   VAR
      sFB_ParaAcycRead { ExternalAccessible := 'False'; ExternalVisible := 'False'; ExternalWritable := 'False'; S7_SetPoint := 'False'} : "FB_VfdNORDParaAcycRead";
      sFB_ParaAcycWrite { ExternalAccessible := 'False'; ExternalVisible := 'False'; ExternalWritable := 'False'; S7_SetPoint := 'False'} : "FB_VfdNORDParaAcycWrite";
      sR_TRIG_Done {InstructionName := 'R_TRIG'; LibVersion := '1.0'; ExternalAccessible := 'False'; ExternalVisible := 'False'; ExternalWritable := 'False'; S7_SetPoint := 'False'} : R_TRIG;
      sR_TRIG_StartJob {InstructionName := 'R_TRIG'; LibVersion := '1.0'; ExternalAccessible := 'False'; ExternalVisible := 'False'; ExternalWritable := 'False'; S7_SetPoint := 'False'} : R_TRIG;   // Bit for start trigger for rising edge
      sF_TRIG_CancelJob {InstructionName := 'F_TRIG'; LibVersion := '1.0'; ExternalAccessible := 'False'; ExternalVisible := 'False'; ExternalWritable := 'False'; S7_SetPoint := 'False'} : F_TRIG;   // Bit for start trigger for falling edge
      sa_Parameter { ExternalAccessible := 'False'; ExternalVisible := 'False'; ExternalWritable := 'False'; S7_SetPoint := 'False'} : Array[0..60] of "UDT_VfdNordParameter";   // Data of parameters
      sa_Status { ExternalAccessible := 'False'; ExternalVisible := 'False'; ExternalWritable := 'False'} : Struct   // Parametrization status
         StepNrError { ExternalAccessible := 'False'; ExternalVisible := 'False'; ExternalWritable := 'False'} : Int;   // The number of the step in witch the error occurred
         ParameterNrError { ExternalAccessible := 'False'; ExternalVisible := 'False'; ExternalWritable := 'False'} : Int;   // The number of the parameter in witch the error occurred
         StepNr { ExternalAccessible := 'False'; ExternalVisible := 'False'; ExternalWritable := 'False'} : Int := 0;   // Current step number
         ResponseValueError { ExternalAccessible := 'False'; ExternalVisible := 'False'; ExternalWritable := 'False'} : Bool;   // Response value error
         WrongFormat { ExternalAccessible := 'False'; ExternalVisible := 'False'; ExternalWritable := 'False'} : Bool;   // Wrong parameter format
         TimeExceeded { ExternalAccessible := 'False'; ExternalVisible := 'False'; ExternalWritable := 'False'} : Bool;   // Time has been exceeded
         NeedAck { ExternalAccessible := 'False'; ExternalVisible := 'False'; ExternalWritable := 'False'} : Bool;   // Need acknowledge signal (to cintinue parametrization)
         StepDone { ExternalAccessible := 'False'; ExternalVisible := 'False'; ExternalWritable := 'False'} : Bool;   // Step done
      END_STRUCT;
      si_StepTime { ExternalAccessible := 'False'; ExternalVisible := 'False'; ExternalWritable := 'False'} : Int;
      si_StepMax { ExternalAccessible := 'False'; ExternalVisible := 'False'; ExternalWritable := 'False'} : Int := 0;   // Maximum step number
      sx_Start { ExternalAccessible := 'False'; ExternalVisible := 'False'; ExternalWritable := 'False'} : Bool;   // Signal to start of parameterization function SinaPara
      sx_Busy { ExternalAccessible := 'False'; ExternalVisible := 'False'; ExternalWritable := 'False'} : Bool;   // Parametrization in progress (busy)
      sx_Done { ExternalAccessible := 'False'; ExternalVisible := 'False'; ExternalWritable := 'False'} : Bool;   // Parametrization done
      sx_Error { ExternalAccessible := 'False'; ExternalVisible := 'False'; ExternalWritable := 'False'} : Bool;   // Main error signal
      sx_PreparedData { ExternalAccessible := 'False'; ExternalVisible := 'False'; ExternalWritable := 'False'} : Bool;   // Step data prepared
      sx_ReadOrder { ExternalAccessible := 'False'; ExternalVisible := 'False'; ExternalWritable := 'False'} : Bool;   // Order to read paraeter with transition from 0 to 1
      sx_WriteOrder { ExternalAccessible := 'False'; ExternalVisible := 'False'; ExternalWritable := 'False'} : Bool;   // Order to write parameter with transition from 0 to 1
      sx_MaxStepCalculation { ExternalAccessible := 'False'; ExternalVisible := 'False'; ExternalWritable := 'False'} : Bool;   // Maximum step calculated
   END_VAR
   VAR RETAIN
      sx_24VCommissioningDone { ExternalAccessible := 'False'; ExternalVisible := 'False'; ExternalWritable := 'False'} : Bool;   // 24V commissioning done succesfully
   END_VAR

   VAR_TEMP
      ti_index : Int;   // Temporary array index
      ti_ControlMethod : Int;
      ti_EncoderCode : Int;
      ti_i : Int;   // Loop counter
      ti_BrakeReaction : Int;
   END_VAR

   VAR CONSTANT
      ci_CFC_ClosedLoop : Int := 1;
      ci_CFC_OpenLoop : Int := 0;
      ci_EncoderRes512 : Int := 1;
      ci_EncoderRes1024 : Int := 3;
      ci_EncoderRes2048 : Int := 5;
      ci_EncoderRes4096 : Int := 6;
      ci_MaxStepTime : Int := 100;
   END_VAR


BEGIN
	(*
	----------------------------------------------------------------------------------------

	Version history:
	Date        | Version   | Author        | Remark
	----------------------------------------------------------------------------------------
	12/01/2020  | 0.1       | S.Theocharis  | Initial version TIA 15.1
	08/04/2021  | 0.2       | F.Baten       | New read/write blocks
	                                        | New motor parameter set ( most values not 32bit )
	                                        | PN device with onboard safety
	                                        | Reading and writing optimised
	27/01/2022  | 0.3       | K.Pokorski    | Add 24V and 400V commissionig status
	                                        | Fix VFD Output bug
	                                        | Initialize InUse status in all parameters
	                                        | Fix Motor identification
	                                        | Save parameters to External memory
	                                        | Delete saving F-parameters from sequence (not working and creating faults)
	                                        | Delete reading CRC code (reading old CRC code what can be confusing)
	21/04/2022  | 0.4       | K.Pokorski    | Delete motor identification
	21/02/2023  | 4.0       | F.Baten       | 4.0 Release TIA 17.5

	*)

	REGION 1 - Start Job

	    // Monitor rising trigger if is input enable signal
	    #sR_TRIG_StartJob(CLK := #iqx_Enable);

	    IF (#sR_TRIG_StartJob.Q)
	    THEN
	        #sx_Start := TRUE;
	        #sx_Busy := TRUE;
	        #sx_Done := FALSE;
	        #sx_Error := FALSE;
	        #sx_PreparedData := FALSE;
	        #sx_MaxStepCalculation := FALSE;
	        #sa_Status.StepDone := FALSE;
	        #sa_Status.StepNrError := 0;
	        #sa_Status.ParameterNrError := 0;
	        #sa_Status.StepNr := 0;
	        #si_StepTime := 0;
	        #qi_HWAdress := 0;

	        FOR #ti_i := 0 TO 60 DO
	            #sa_Parameter[#ti_i].InUse := FALSE;
	        END_FOR;



	    END_IF;

	END_REGION

	REGION 2 - Build Sequences in static memory

	    IF #sR_TRIG_StartJob.Q THEN
	        //  IF NOT #sx_24VCommissioningDone THEN
	        REGION Step 01 - P523 Factory reset [0..3]
	            #ti_index := 0;
	            #sa_Parameter[#ti_index].ParaNumber := 523;
	            #sa_Parameter[#ti_index].Index := 0;
	            #sa_Parameter[#ti_index].WriteValue := 1;
	            #sa_Parameter[#ti_index].WriteAccess := TRUE;
	            #sa_Parameter[#ti_index].ParaSet := 0;
	            #sa_Parameter[#ti_index].Format32 := FALSE;
	            #sa_Parameter[#ti_index].ActualValue := 0;
	            #sa_Parameter[#ti_index].InUse := TRUE;
	            #sa_Parameter[#ti_index].RamOnly := FALSE;
	        END_REGION

	        REGION Step 02 - P003 Set supervisor code to access all parameters [0..9999]
	            #ti_index := #ti_index + 1;
	            #sa_Parameter[#ti_index].ParaNumber := 3;
	            #sa_Parameter[#ti_index].Index := 0;
	            #sa_Parameter[#ti_index].WriteValue := 3;
	            #sa_Parameter[#ti_index].WriteAccess := TRUE;
	            #sa_Parameter[#ti_index].ParaSet := 0;
	            #sa_Parameter[#ti_index].Format32 := FALSE;
	            #sa_Parameter[#ti_index].ActualValue := 0;
	            #sa_Parameter[#ti_index].InUse := TRUE;
	            #sa_Parameter[#ti_index].RamOnly := FALSE;
	        END_REGION

	        REGION Step 03 - P800 Set Operating mode Safety [0-1]
	            #ti_index := #ti_index + 1;
	            #sa_Parameter[#ti_index].ParaNumber := 800;
	            #sa_Parameter[#ti_index].Index := 1;
	            #sa_Parameter[#ti_index].WriteValue := 1;
	            #sa_Parameter[#ti_index].WriteAccess := TRUE;
	            #sa_Parameter[#ti_index].ParaSet := 0;
	            #sa_Parameter[#ti_index].Format32 := FALSE;
	            #sa_Parameter[#ti_index].ActualValue := 0;
	            #sa_Parameter[#ti_index].InUse := TRUE;
	            #sa_Parameter[#ti_index].RamOnly := FALSE;
	        END_REGION

	        REGION Step 04 - P800 Set Operating mode Safety [0-1]
	            #ti_index := #ti_index + 1;
	            #sa_Parameter[#ti_index].ParaNumber := 800;
	            #sa_Parameter[#ti_index].Index := 2;
	            #sa_Parameter[#ti_index].WriteValue := 0;
	            #sa_Parameter[#ti_index].WriteAccess := TRUE;
	            #sa_Parameter[#ti_index].ParaSet := 0;
	            #sa_Parameter[#ti_index].Format32 := FALSE;
	            #sa_Parameter[#ti_index].ActualValue := 0;
	            #sa_Parameter[#ti_index].InUse := TRUE;
	            #sa_Parameter[#ti_index].RamOnly := FALSE;
	        END_REGION

	        REGION Step 05 - P802 Set Enable safety channel [0-1]  Channel 1 on
	            #ti_index := #ti_index + 1;
	            #sa_Parameter[#ti_index].ParaNumber := 802;
	            #sa_Parameter[#ti_index].Index := 1;
	            #sa_Parameter[#ti_index].WriteValue := 1;
	            #sa_Parameter[#ti_index].WriteAccess := TRUE;
	            #sa_Parameter[#ti_index].ParaSet := 0;
	            #sa_Parameter[#ti_index].Format32 := FALSE;
	            #sa_Parameter[#ti_index].ActualValue := 0;
	            #sa_Parameter[#ti_index].InUse := TRUE;
	            #sa_Parameter[#ti_index].RamOnly := FALSE;
	        END_REGION

	        REGION Step 06 - P802 Set Enable safety channel [0-1]  Channel 2 on
	            #ti_index := #ti_index + 1;
	            #sa_Parameter[#ti_index].ParaNumber := 802;
	            #sa_Parameter[#ti_index].Index := 2;
	            #sa_Parameter[#ti_index].WriteValue := 1;
	            #sa_Parameter[#ti_index].WriteAccess := TRUE;
	            #sa_Parameter[#ti_index].ParaSet := 0;
	            #sa_Parameter[#ti_index].Format32 := FALSE;
	            #sa_Parameter[#ti_index].ActualValue := 0;
	            #sa_Parameter[#ti_index].InUse := TRUE;
	            #sa_Parameter[#ti_index].RamOnly := FALSE;
	        END_REGION

	        REGION Step 07 - P802 Set Enable safety channel [0-1]  Channel 3 on
	            #ti_index := #ti_index + 1;
	            #sa_Parameter[#ti_index].ParaNumber := 802;
	            #sa_Parameter[#ti_index].Index := 3;
	            #sa_Parameter[#ti_index].WriteValue := 1;
	            #sa_Parameter[#ti_index].WriteAccess := TRUE;
	            #sa_Parameter[#ti_index].ParaSet := 0;
	            #sa_Parameter[#ti_index].Format32 := FALSE;
	            #sa_Parameter[#ti_index].ActualValue := 0;
	            #sa_Parameter[#ti_index].InUse := TRUE;
	            #sa_Parameter[#ti_index].RamOnly := FALSE;
	        END_REGION

	        REGION Step 08 - P846 Read dipswitches
	            #ti_index := #ti_index + 1;
	            #sa_Parameter[#ti_index].ParaNumber := 846;
	            #sa_Parameter[#ti_index].Index := 0;
	            #sa_Parameter[#ti_index].WriteValue := 0;
	            #sa_Parameter[#ti_index].WriteAccess := FALSE;
	            #sa_Parameter[#ti_index].ParaSet := 0;
	            #sa_Parameter[#ti_index].Format32 := FALSE;
	            #sa_Parameter[#ti_index].ActualValue := 0;
	            #sa_Parameter[#ti_index].InUse := TRUE;
	            #sa_Parameter[#ti_index].RamOnly := FALSE;
	        END_REGION

	        REGION Step 09 - P120 Set extern control units [0-1]  Switch off 3 and 4
	            #ti_index := #ti_index + 1;
	            #sa_Parameter[#ti_index].ParaNumber := 120;
	            #sa_Parameter[#ti_index].Index := 3;
	            #sa_Parameter[#ti_index].WriteValue := 0;
	            #sa_Parameter[#ti_index].WriteAccess := TRUE;
	            #sa_Parameter[#ti_index].ParaSet := 0;
	            #sa_Parameter[#ti_index].Format32 := FALSE;
	            #sa_Parameter[#ti_index].ActualValue := 0;
	            #sa_Parameter[#ti_index].InUse := TRUE;
	            #sa_Parameter[#ti_index].RamOnly := FALSE;
	        END_REGION

	        REGION Step 10 - P120 Set extern control units [0-1]  Switch off 3 and 4
	            #ti_index := #ti_index + 1;
	            #sa_Parameter[#ti_index].ParaNumber := 120;
	            #sa_Parameter[#ti_index].Index := 4;
	            #sa_Parameter[#ti_index].WriteValue := 0;
	            #sa_Parameter[#ti_index].WriteAccess := TRUE;
	            #sa_Parameter[#ti_index].ParaSet := 0;
	            #sa_Parameter[#ti_index].Format32 := FALSE;
	            #sa_Parameter[#ti_index].ActualValue := 0;
	            #sa_Parameter[#ti_index].InUse := TRUE;
	            #sa_Parameter[#ti_index].RamOnly := FALSE;
	        END_REGION

	        REGION Step 11 - P202 Write motor nominal speed [150...24000]rpm
	            #ti_index := #ti_index + 1;
	            #sa_Parameter[#ti_index].ParaNumber := 202;
	            #sa_Parameter[#ti_index].Index := 0;
	            #sa_Parameter[#ti_index].WriteValue := #iudt_MotorData.NominalSpeed;
	            #sa_Parameter[#ti_index].WriteAccess := TRUE;
	            #sa_Parameter[#ti_index].ParaSet := 1; // Parameter set 1
	            #sa_Parameter[#ti_index].Format32 := FALSE;
	            #sa_Parameter[#ti_index].ActualValue := 0;
	            #sa_Parameter[#ti_index].InUse := TRUE;
	            #sa_Parameter[#ti_index].RamOnly := FALSE;
	        END_REGION

	        REGION Step 12 - P203 Write motor nominal current [0.1 ...1000.0]A
	            #ti_index := #ti_index + 1;
	            #sa_Parameter[#ti_index].ParaNumber := 203;
	            #sa_Parameter[#ti_index].Index := 0;
	            #sa_Parameter[#ti_index].WriteValue := (REAL_TO_DINT(#iudt_MotorData.NominalCurrent * 10));  // Value 55 = 5.5 Amps
	            #sa_Parameter[#ti_index].WriteAccess := TRUE;
	            #sa_Parameter[#ti_index].ParaSet := 0; // Parameter set 1
	            #sa_Parameter[#ti_index].Format32 := FALSE;
	            #sa_Parameter[#ti_index].ActualValue := 0;
	            #sa_Parameter[#ti_index].InUse := TRUE;
	            #sa_Parameter[#ti_index].RamOnly := FALSE;
	        END_REGION

	        REGION Step 13 - P204 Write motor nominal voltage [100 ... 800]V
	            #ti_index := #ti_index + 1;
	            #sa_Parameter[#ti_index].ParaNumber := 204;
	            #sa_Parameter[#ti_index].Index := 0;
	            #sa_Parameter[#ti_index].WriteValue := #iudt_MotorData.NominalVoltage;
	            #sa_Parameter[#ti_index].WriteAccess := FALSE;
	            #sa_Parameter[#ti_index].ParaSet := 1; // Parameter set 1
	            #sa_Parameter[#ti_index].Format32 := FALSE;
	            #sa_Parameter[#ti_index].ActualValue := 0;
	            #sa_Parameter[#ti_index].InUse := TRUE;
	            #sa_Parameter[#ti_index].RamOnly := FALSE;
	        END_REGION

	        REGION Step 14 - P205 Write motor nominal power
	            #ti_index := #ti_index + 1;
	            #sa_Parameter[#ti_index].ParaNumber := 205;
	            #sa_Parameter[#ti_index].Index := 0;
	            #sa_Parameter[#ti_index].WriteValue := (REAL_TO_DINT(#iudt_MotorData.NominalPower * 100));
	            #sa_Parameter[#ti_index].WriteAccess := TRUE;
	            #sa_Parameter[#ti_index].ParaSet := 0; // Parameter set 1
	            #sa_Parameter[#ti_index].Format32 := FALSE;
	            #sa_Parameter[#ti_index].ActualValue := 0;
	            #sa_Parameter[#ti_index].InUse := TRUE;
	            #sa_Parameter[#ti_index].RamOnly := FALSE;
	        END_REGION

	        REGION Step 15 - P206 Write motor cosPhi [0.50 ... 0.95]
	            #ti_index := #ti_index + 1;
	            #sa_Parameter[#ti_index].ParaNumber := 206;
	            #sa_Parameter[#ti_index].Index := 0;
	            #sa_Parameter[#ti_index].WriteValue := REAL_TO_DINT(#iudt_MotorData.CosPhi * 100);
	            #sa_Parameter[#ti_index].WriteAccess := TRUE;
	            #sa_Parameter[#ti_index].ParaSet := 0; // Parameter set 1
	            #sa_Parameter[#ti_index].Format32 := FALSE;
	            #sa_Parameter[#ti_index].ActualValue := 0;
	            #sa_Parameter[#ti_index].InUse := TRUE;
	            #sa_Parameter[#ti_index].RamOnly := FALSE;
	        END_REGION

	        REGION Step 16 - P207 Connection Star / Delta [0=Star 1=Delta]
	            #ti_index := #ti_index + 1;
	            #sa_Parameter[#ti_index].ParaNumber := 207;
	            #sa_Parameter[#ti_index].Index := 0;
	            #sa_Parameter[#ti_index].WriteValue := #iudt_MotorData.Connection;
	            #sa_Parameter[#ti_index].WriteAccess := TRUE;
	            #sa_Parameter[#ti_index].ParaSet := 0; // Parameter set 1
	            #sa_Parameter[#ti_index].Format32 := FALSE;
	            #sa_Parameter[#ti_index].ActualValue := 0;
	            #sa_Parameter[#ti_index].InUse := TRUE;
	            #sa_Parameter[#ti_index].RamOnly := FALSE;
	        END_REGION

	        REGION Step 17 - P105 Write Maximum / Reference Frequency [0.1...400.0]Hz
	            #ti_index := #ti_index + 1;
	            #sa_Parameter[#ti_index].ParaNumber := 105;
	            #sa_Parameter[#ti_index].Index := 0;
	            #sa_Parameter[#ti_index].WriteValue := REAL_TO_DINT(#ir_ReferenceFrequency * 10);
	            #sa_Parameter[#ti_index].WriteAccess := TRUE;
	            #sa_Parameter[#ti_index].ParaSet := 0; // Parameter set 1
	            #sa_Parameter[#ti_index].Format32 := FALSE;
	            #sa_Parameter[#ti_index].ActualValue := 0;
	            #sa_Parameter[#ti_index].InUse := TRUE;
	            #sa_Parameter[#ti_index].RamOnly := FALSE;
	        END_REGION

	        REGION Step 18 - P107 Brake reaction
	            IF #iudt_MotorData.BrakeConfig THEN
	                #ti_BrakeReaction := 20;
	            ELSE
	                #ti_BrakeReaction := 0;
	            END_IF;

	            #ti_index := #ti_index + 1;
	            #sa_Parameter[#ti_index].ParaNumber := 107;
	            #sa_Parameter[#ti_index].Index := 0;
	            #sa_Parameter[#ti_index].WriteValue := #ti_BrakeReaction;
	            #sa_Parameter[#ti_index].WriteAccess := TRUE;
	            #sa_Parameter[#ti_index].ParaSet := 0; // Parameter set 1
	            #sa_Parameter[#ti_index].Format32 := FALSE;
	            #sa_Parameter[#ti_index].ActualValue := 0;
	            #sa_Parameter[#ti_index].InUse := TRUE;
	            #sa_Parameter[#ti_index].RamOnly := FALSE;
	        END_REGION

	        REGION Step 19 - P300 Mode [0..2]
	            //If an IE4 motor is operated in CFC closed loop mode , the slip error monitoring must be activated. P327<>0
	            IF #iudt_MotorData.EncoderResolution <> 0 THEN
	                #ti_ControlMethod := #ci_CFC_ClosedLoop; //CFC closed loop control. Speed control with encoder feedback
	            ELSE
	                #ti_ControlMethod := #ci_CFC_OpenLoop; //VFC open loop control. Speed control without encoder feedback
	            END_IF;
	            #ti_index := #ti_index + 1;
	            #sa_Parameter[#ti_index].ParaNumber := 300;
	            #sa_Parameter[#ti_index].Index := 0;
	            #sa_Parameter[#ti_index].WriteValue := #ti_ControlMethod;
	            #sa_Parameter[#ti_index].WriteAccess := TRUE;
	            #sa_Parameter[#ti_index].ParaSet := 1; // Parameter set 1
	            #sa_Parameter[#ti_index].Format32 := FALSE;
	            #sa_Parameter[#ti_index].ActualValue := 0;
	            #sa_Parameter[#ti_index].InUse := TRUE;
	            #sa_Parameter[#ti_index].RamOnly := FALSE;
	        END_REGION

	        REGION Step 20 - P301 Encoder Resolution [0..17]
	            CASE #iudt_MotorData.EncoderResolution OF
	                512:
	                    #ti_EncoderCode := #ci_EncoderRes512;
	                1024:
	                    #ti_EncoderCode := #ci_EncoderRes1024;
	                2048:
	                    #ti_EncoderCode := #ci_EncoderRes2048;
	                4096:
	                    #ti_EncoderCode := #ci_EncoderRes4096;
	                ELSE
	                    #ti_EncoderCode := 6; //default value
	            END_CASE;

	            #ti_index := #ti_index + 1;
	            #sa_Parameter[#ti_index].ParaNumber := 301;
	            #sa_Parameter[#ti_index].Index := 0;
	            #sa_Parameter[#ti_index].WriteValue := #ti_EncoderCode;
	            #sa_Parameter[#ti_index].WriteAccess := TRUE;
	            #sa_Parameter[#ti_index].ParaSet := 0;
	            #sa_Parameter[#ti_index].Format32 := FALSE;
	            #sa_Parameter[#ti_index].ActualValue := 0;
	            #sa_Parameter[#ti_index].InUse := TRUE;
	            #sa_Parameter[#ti_index].RamOnly := FALSE;
	        END_REGION

	        REGION Step 21 - P326 Encoder ratio [0.01 ... 100.0]
	            #ti_index := #ti_index + 1;
	            #sa_Parameter[#ti_index].ParaNumber := 326;
	            #sa_Parameter[#ti_index].Index := 0;
	            #sa_Parameter[#ti_index].WriteValue := (1 * 100); //leave temporary the default 1.00;
	            #sa_Parameter[#ti_index].WriteAccess := TRUE;
	            #sa_Parameter[#ti_index].ParaSet := 0;
	            #sa_Parameter[#ti_index].Format32 := FALSE;
	            #sa_Parameter[#ti_index].ActualValue := 0;
	            #sa_Parameter[#ti_index].InUse := TRUE;
	            #sa_Parameter[#ti_index].RamOnly := FALSE;
	        END_REGION

	        REGION Step 22 - P420[1] Digital inputs [0 ... 80] DI1
	            #ti_index := #ti_index + 1;
	            #sa_Parameter[#ti_index].ParaNumber := 420;
	            #sa_Parameter[#ti_index].Index := 1;
	            #sa_Parameter[#ti_index].WriteValue := 0;
	            #sa_Parameter[#ti_index].WriteAccess := TRUE;
	            #sa_Parameter[#ti_index].ParaSet := 0;
	            #sa_Parameter[#ti_index].Format32 := FALSE;
	            #sa_Parameter[#ti_index].ActualValue := 0;
	            #sa_Parameter[#ti_index].InUse := TRUE;
	            #sa_Parameter[#ti_index].RamOnly := FALSE;
	        END_REGION

	        REGION Step 23 - P420[2] Digital inputs [0 ... 80] DI2
	            #ti_index := #ti_index + 1;
	            #sa_Parameter[#ti_index].ParaNumber := 420;
	            #sa_Parameter[#ti_index].Index := 2;
	            #sa_Parameter[#ti_index].WriteValue := 0;
	            #sa_Parameter[#ti_index].WriteAccess := TRUE;
	            #sa_Parameter[#ti_index].ParaSet := 0;
	            #sa_Parameter[#ti_index].Format32 := FALSE;
	            #sa_Parameter[#ti_index].ActualValue := 0;
	            #sa_Parameter[#ti_index].InUse := TRUE;
	            #sa_Parameter[#ti_index].RamOnly := FALSE;
	        END_REGION

	        REGION Step 24 - P420[3] Digital inputs [0 ... 80] DI3
	            #ti_index := #ti_index + 1;
	            #sa_Parameter[#ti_index].ParaNumber := 420;
	            #sa_Parameter[#ti_index].Index := 3;
	            #sa_Parameter[#ti_index].WriteValue := 0;
	            #sa_Parameter[#ti_index].WriteAccess := TRUE;
	            #sa_Parameter[#ti_index].ParaSet := 0;
	            #sa_Parameter[#ti_index].Format32 := FALSE;
	            #sa_Parameter[#ti_index].ActualValue := 0;
	            #sa_Parameter[#ti_index].InUse := TRUE;
	            #sa_Parameter[#ti_index].RamOnly := FALSE;
	        END_REGION

	        REGION Step 25 - P426 Quick Stop time [0 ... 320.00] sec
	            #ti_index := #ti_index + 1;
	            #sa_Parameter[#ti_index].ParaNumber := 426;
	            #sa_Parameter[#ti_index].Index := 0;
	            #sa_Parameter[#ti_index].WriteValue := 60;
	            #sa_Parameter[#ti_index].WriteAccess := TRUE;
	            #sa_Parameter[#ti_index].ParaSet := 1; //paraset 1
	            #sa_Parameter[#ti_index].Format32 := FALSE;
	            #sa_Parameter[#ti_index].ActualValue := 0;
	            #sa_Parameter[#ti_index].InUse := TRUE;
	            #sa_Parameter[#ti_index].RamOnly := FALSE;
	        END_REGION

	        REGION Step 26 - P509 Control word source [0..4]
	            #ti_index := #ti_index + 1;
	            #sa_Parameter[#ti_index].ParaNumber := 509;
	            #sa_Parameter[#ti_index].Index := 0;
	            #sa_Parameter[#ti_index].WriteValue := 3; // System bus communication (PN)
	            #sa_Parameter[#ti_index].WriteAccess := TRUE;
	            #sa_Parameter[#ti_index].ParaSet := 0;
	            #sa_Parameter[#ti_index].Format32 := FALSE;
	            #sa_Parameter[#ti_index].ActualValue := 0;
	            #sa_Parameter[#ti_index].InUse := TRUE;
	            #sa_Parameter[#ti_index].RamOnly := FALSE;
	        END_REGION

	        REGION Step 27 - P543[1] Actual speed to actual value 1 [0..57]
	            #ti_index := #ti_index + 1;
	            #sa_Parameter[#ti_index].ParaNumber := 543;
	            #sa_Parameter[#ti_index].Index := 1;
	            #sa_Parameter[#ti_index].WriteValue := 1; // 2 = Set Actual value 1 to actual speed
	            #sa_Parameter[#ti_index].WriteAccess := TRUE;
	            #sa_Parameter[#ti_index].ParaSet := 1; // Parameter set 1
	            #sa_Parameter[#ti_index].Format32 := FALSE;
	            #sa_Parameter[#ti_index].ActualValue := 0;
	            #sa_Parameter[#ti_index].InUse := TRUE;
	            #sa_Parameter[#ti_index].RamOnly := FALSE;
	        END_REGION

	        REGION Step 28 - P543[2] Error code to actual value 2 [0..57]
	            #ti_index := #ti_index + 1;
	            #sa_Parameter[#ti_index].ParaNumber := 543;
	            #sa_Parameter[#ti_index].Index := 2;
	            #sa_Parameter[#ti_index].WriteValue := 9; // 9 =  Set Actual value 2 to error code
	            #sa_Parameter[#ti_index].WriteAccess := TRUE;
	            #sa_Parameter[#ti_index].ParaSet := 1; // Parameter set 1
	            #sa_Parameter[#ti_index].Format32 := FALSE;
	            #sa_Parameter[#ti_index].ActualValue := 0;
	            #sa_Parameter[#ti_index].InUse := TRUE;
	            #sa_Parameter[#ti_index].RamOnly := FALSE;
	        END_REGION

	        REGION Step 29 - P543[3] DIO status to actual value 3 [0..57]
	            #ti_index := #ti_index + 1;
	            #sa_Parameter[#ti_index].ParaNumber := 543;
	            #sa_Parameter[#ti_index].Index := 3;
	            #sa_Parameter[#ti_index].WriteValue := 5; // 5 =  Set Actual value 3 to DIO status
	            #sa_Parameter[#ti_index].WriteAccess := TRUE;
	            #sa_Parameter[#ti_index].ParaSet := 1; // Parameter set 1
	            #sa_Parameter[#ti_index].Format32 := FALSE;
	            #sa_Parameter[#ti_index].ActualValue := 0;
	            #sa_Parameter[#ti_index].InUse := TRUE;
	            #sa_Parameter[#ti_index].RamOnly := FALSE;
	        END_REGION

	        REGION Step 30 - P546[1] Frequency setpoint to setpoint 1 [0..36]
	            #ti_index := #ti_index + 1;
	            #sa_Parameter[#ti_index].ParaNumber := 546;
	            #sa_Parameter[#ti_index].Index := 1;
	            #sa_Parameter[#ti_index].WriteValue := 1; // 5 =  Set setpoint 1 to frequency setpoint
	            #sa_Parameter[#ti_index].WriteAccess := TRUE;
	            #sa_Parameter[#ti_index].ParaSet := 1; // Parameter set 1
	            #sa_Parameter[#ti_index].Format32 := FALSE;
	            #sa_Parameter[#ti_index].ActualValue := 0;
	            #sa_Parameter[#ti_index].InUse := TRUE;
	            #sa_Parameter[#ti_index].RamOnly := FALSE;
	        END_REGION

	        REGION Step 31 - P546[2] Ramp setpoint to setpoint 2 [0..36]
	            #ti_index := #ti_index + 1;
	            #sa_Parameter[#ti_index].ParaNumber := 546;
	            #sa_Parameter[#ti_index].Index := 2;
	            #sa_Parameter[#ti_index].WriteValue := 15; // 15 =  Set setpoint 2 to ramp setpoint
	            #sa_Parameter[#ti_index].WriteAccess := TRUE;
	            #sa_Parameter[#ti_index].ParaSet := 1; // Parameter set 1
	            #sa_Parameter[#ti_index].Format32 := FALSE;
	            #sa_Parameter[#ti_index].ActualValue := 0;
	            #sa_Parameter[#ti_index].InUse := TRUE;
	            #sa_Parameter[#ti_index].RamOnly := FALSE;
	        END_REGION

	        REGION Step 32 - P546[3] DO control to setpoint 3 [0..36]
	            #ti_index := #ti_index + 1;
	            #sa_Parameter[#ti_index].ParaNumber := 546;
	            #sa_Parameter[#ti_index].Index := 3;
	            #sa_Parameter[#ti_index].WriteValue := 31; // 5 =  Set setpoint 3 to DIO
	            #sa_Parameter[#ti_index].WriteAccess := TRUE;
	            #sa_Parameter[#ti_index].ParaSet := 1; // Parameter set 1
	            #sa_Parameter[#ti_index].Format32 := FALSE;
	            #sa_Parameter[#ti_index].ActualValue := 0;
	            #sa_Parameter[#ti_index].InUse := TRUE;
	            #sa_Parameter[#ti_index].RamOnly := FALSE;
	        END_REGION

	        REGION Step 33 - P434[3] DO Function [1..2]
	            #ti_index := #ti_index + 1;
	            #sa_Parameter[#ti_index].ParaNumber := 434;
	            #sa_Parameter[#ti_index].Index := 1;
	            #sa_Parameter[#ti_index].WriteValue := 38;
	            #sa_Parameter[#ti_index].WriteAccess := TRUE;
	            #sa_Parameter[#ti_index].ParaSet := 1; // Parameter set 1
	            #sa_Parameter[#ti_index].Format32 := FALSE;
	            #sa_Parameter[#ti_index].ActualValue := 0;
	            #sa_Parameter[#ti_index].InUse := TRUE;
	            #sa_Parameter[#ti_index].RamOnly := FALSE;
	        END_REGION

	        REGION Step 34 - P560 Save [0..2]
	            #ti_index := #ti_index + 1;
	            #sa_Parameter[#ti_index].ParaNumber := 560;
	            #sa_Parameter[#ti_index].Index := 0;
	            #sa_Parameter[#ti_index].WriteValue := 1; // 1= save RAM & EERPOM
	            #sa_Parameter[#ti_index].WriteAccess := TRUE;
	            #sa_Parameter[#ti_index].ParaSet := 0;
	            #sa_Parameter[#ti_index].Format32 := FALSE;
	            #sa_Parameter[#ti_index].ActualValue := 0;
	            #sa_Parameter[#ti_index].InUse := TRUE;
	            #sa_Parameter[#ti_index].RamOnly := FALSE;
	        END_REGION

	        REGION Step 35 - P550 Copy internal EEPROM to external EEPROM [0..3]
	            #ti_index := #ti_index + 1;
	            #sa_Parameter[#ti_index].ParaNumber := 550;
	            #sa_Parameter[#ti_index].Index := 0;
	            #sa_Parameter[#ti_index].WriteValue := 2; // 2 = Copy internal to external EEPROM
	            #sa_Parameter[#ti_index].WriteAccess := FALSE;
	            #sa_Parameter[#ti_index].ParaSet := 0;
	            #sa_Parameter[#ti_index].Format32 := FALSE;
	            #sa_Parameter[#ti_index].ActualValue := 0;
	            #sa_Parameter[#ti_index].InUse := TRUE;
	            #sa_Parameter[#ti_index].RamOnly := FALSE;
	        END_REGION
	    END_IF;

	    (* IF #ix_VFDReadyToRun AND #sx_24VCommissioningDone THEN
	         REGION Step 39 - P220 Measurement [0..2]
	             #ti_index := 0;
	             #sa_Parameter[#ti_index].ParaNumber := 220;
	             #sa_Parameter[#ti_index].Index := 0;
	             #sa_Parameter[#ti_index].WriteValue := 2; // 2 =  Motor identification
	             #sa_Parameter[#ti_index].WriteAccess := TRUE;
	             #sa_Parameter[#ti_index].ParaSet := 1;
	             #sa_Parameter[#ti_index].Format32 := FALSE;
	             #sa_Parameter[#ti_index].ActualValue := 0;
	             #sa_Parameter[#ti_index].InUse := TRUE;
	             #sa_Parameter[#ti_index].RamOnly := FALSE;
	         END_REGION

	         REGION Step 40 - P220 Read if measurement started
	             #ti_index := #ti_index + 1;
	             #sa_Parameter[#ti_index].ParaNumber := 220;
	             #sa_Parameter[#ti_index].Index := 0;
	             #sa_Parameter[#ti_index].WriteValue := 0;
	             #sa_Parameter[#ti_index].WriteAccess := FALSE;
	             #sa_Parameter[#ti_index].ParaSet := 1;
	             #sa_Parameter[#ti_index].Format32 := FALSE;
	             #sa_Parameter[#ti_index].ActualValue := 0;
	             #sa_Parameter[#ti_index].InUse := TRUE;
	             #sa_Parameter[#ti_index].RamOnly := FALSE;
	         END_REGION

	         REGION Step 41 - P220 Read if measurement finished
	             #ti_index := #ti_index + 1;
	             #sa_Parameter[#ti_index].ParaNumber := 220;
	             #sa_Parameter[#ti_index].Index := 0;
	             #sa_Parameter[#ti_index].WriteValue := 0;
	             #sa_Parameter[#ti_index].WriteAccess := FALSE;
	             #sa_Parameter[#ti_index].ParaSet := 1;
	             #sa_Parameter[#ti_index].Format32 := FALSE;
	             #sa_Parameter[#ti_index].ActualValue := 0;
	             #sa_Parameter[#ti_index].InUse := TRUE;
	             #sa_Parameter[#ti_index].RamOnly := FALSE;
	         END_REGION


	         REGION Step 42 - P560 Save [0..2] (Step 39 - without motor identification)
	             #ti_index := #ti_index + 1;
	             #sa_Parameter[#ti_index].ParaNumber := 560;
	             #sa_Parameter[#ti_index].Index := 0;
	             #sa_Parameter[#ti_index].WriteValue := 1; // 1= save RAM & EERPOM
	             #sa_Parameter[#ti_index].WriteAccess := TRUE;
	             #sa_Parameter[#ti_index].ParaSet := 0;
	             #sa_Parameter[#ti_index].Format32 := FALSE;
	             #sa_Parameter[#ti_index].ActualValue := 0;
	             #sa_Parameter[#ti_index].InUse := TRUE;
	             #sa_Parameter[#ti_index].RamOnly := FALSE;
	         END_REGION

	         REGION Step 43 - P550 Copy internal EEPROM to external EEPROM [0..3] (Step 40 - without motor identification)
	             #ti_index := #ti_index + 1;
	             #sa_Parameter[#ti_index].ParaNumber := 550;
	             #sa_Parameter[#ti_index].Index := 0;
	             #sa_Parameter[#ti_index].WriteValue := 2; // 2 = Copy internal to external EEPROM
	             #sa_Parameter[#ti_index].WriteAccess := FALSE;
	             #sa_Parameter[#ti_index].ParaSet := 0;
	             #sa_Parameter[#ti_index].Format32 := FALSE;
	             #sa_Parameter[#ti_index].ActualValue := 0;
	             #sa_Parameter[#ti_index].InUse := TRUE;
	             #sa_Parameter[#ti_index].RamOnly := FALSE;
	         END_REGION
	         #sx_MotorMeasurement := TRUE;

	     END_IF; *)

	    // END_IF;

	END_REGION

	REGION 3 - Cancel job

	    // Monitor falling trigger if is input enable signal
	    #sF_TRIG_CancelJob(CLK := #iqx_Enable);

	    IF (#sF_TRIG_CancelJob.Q)
	    THEN
	        // IF parametrization is NOT done
	        IF (NOT #sx_Done)
	        THEN

	            #sx_Error := TRUE;
	            #sx_ReadOrder := FALSE;
	            #sx_WriteOrder := FALSE;
	            #sFB_ParaAcycWrite.qx_Done := FALSE;
	            #sx_Start := FALSE;
	            #sx_Busy := FALSE;

	        END_IF;

	    END_IF;

	END_REGION

	REGION 4 - Caclulaton used step in the sequence
	    // If maximum step is not calculated and input enable signal
	    IF (NOT #sx_MaxStepCalculation
	        AND #iqx_Enable)
	    THEN

	        // Create loop from maximum step number = 1 to 80
	        FOR #si_StepMax := 1 TO 80 DO

	            IF (NOT #sa_Parameter[#si_StepMax].InUse)   // If step commissioning is not used in sequence
	            THEN
	                #sx_MaxStepCalculation := TRUE;
	                EXIT;
	            END_IF;
	        END_FOR;
	    END_IF;
	END_REGION

	REGION 5 - Prepare data

	    IF (#sx_Start                                       // If occurs: signal to start of parametrization
	        AND NOT #sx_PreparedData                        // And step data is not prepared
	        AND NOT #sa_Status.StepDone                      // And parametrization is not done
	        AND #iqx_Enable)                                // And input enable signal
	    THEN

	        #sx_WriteOrder := #sa_Parameter[#sa_Status.StepNr].WriteAccess;
	        #sx_ReadOrder := NOT #sa_Parameter[#sa_Status.StepNr].WriteAccess;
	        #sx_PreparedData := TRUE;

	    END_IF;
	END_REGION

	REGION 6 - Call write parameter block

	    IF #sx_WriteOrder AND #sx_PreparedData THEN
	        #sFB_ParaAcycWrite(HW_Identifier := #ihw_HardwareID,
	                           idi_Value := #sa_Parameter[#sa_Status.StepNr].WriteValue,
	                           ii_ParameterNumber := #sa_Parameter[#sa_Status.StepNr].ParaNumber,
	                           ii_ParameterIndex := #sa_Parameter[#sa_Status.StepNr].Index,
	                           ii_ParameterSet := #sa_Parameter[#sa_Status.StepNr].ParaSet,
	                           ix_Parameter32Bit := #sa_Parameter[#sa_Status.StepNr].Format32,
	                           ix_RAM_Only := #sa_Parameter[#sa_Status.StepNr].RamOnly,
	                           ix_Execute := NOT #sFB_ParaAcycWrite.qx_Done,
	                           qx_Done => #sFB_ParaAcycWrite.qx_Done,
	                           qx_Busy => #sFB_ParaAcycWrite.qx_Busy,
	                           qx_Error => #sFB_ParaAcycWrite.qx_Error,
	                           qdi_ValueRead => #sa_Parameter[#sa_Status.StepNr].ActualValue,
	                           qw_ErrorID => #sFB_ParaAcycWrite.qw_ErrorID);

	        #sR_TRIG_Done(CLK := #sFB_ParaAcycWrite.qx_Done);
	    END_IF;
	END_REGION

	REGION 7 - Call read parameter block

	    IF #sx_ReadOrder AND #sx_PreparedData THEN
	        #sFB_ParaAcycRead(iHW_Identifier := #ihw_HardwareID,
	                          ix_Enable := TRUE,
	                          ii_Parameter_Number := #sa_Parameter[#sa_Status.StepNr].ParaNumber,
	                          ii_Parameter_Index := #sa_Parameter[#sa_Status.StepNr].Index,
	                          ii_Parameter_Set := #sa_Parameter[#sa_Status.StepNr].ParaSet,
	                          qx_Valid => #sFB_ParaAcycRead.qx_Valid,
	                          qx_Busy => #sFB_ParaAcycRead.qx_Busy,
	                          qx_Error => #sFB_ParaAcycRead.qx_Error,
	                          qw_Error_ID => #sFB_ParaAcycRead.qw_Error_ID,
	                          qdi_Value => #sFB_ParaAcycRead.qdi_Value);
	    END_IF;
	END_REGION

	REGION 8 - Status commissioning

	    REGION 8.1 Step number error

	        IF (#sx_WriteOrder AND #sFB_ParaAcycWrite.qx_Error)
	            OR
	            (#sx_ReadOrder AND #sFB_ParaAcycRead.qx_Error)
	            OR #sa_Status.TimeExceeded
	        THEN
	            #sx_Start := FALSE;
	            #sx_Error := TRUE;
	            #sx_Done := FALSE;

	            #sx_WriteOrder := FALSE;
	            #sx_ReadOrder := False;
	            #sa_Status.StepNrError := #sa_Status.StepNr;
	        END_IF;
	    END_REGION


	    REGION 8.2 - Read done

	        IF #sx_ReadOrder
	            AND NOT #sFB_ParaAcycRead.qx_Busy
	            AND NOT #sFB_ParaAcycRead.qx_Error
	            AND #sFB_ParaAcycRead.qx_Valid

	        THEN

	            #sa_Status.StepDone := TRUE;
	            #sx_ReadOrder := FALSE;
	            #sa_Parameter[#sa_Status.StepNr].ActualValue := DINT_TO_INT(#sFB_ParaAcycRead.qdi_Value);

	            IF #sa_Parameter[#sa_Status.StepNr].ParaNumber = 846
	            THEN
	                #qi_HWAdress := DINT_TO_INT(#sFB_ParaAcycRead.qdi_Value);
	            END_IF;

	        END_IF;
	    END_REGION


	    REGION 8.3 - Write done

	        IF #sx_WriteOrder
	            AND NOT #sFB_ParaAcycWrite.qx_Error
	            AND #sR_TRIG_Done.Q
	        THEN
	            #sa_Status.StepDone := TRUE;
	            #sx_WriteOrder := FALSE;
	            #sFB_ParaAcycWrite.qx_Done := FALSE;
	        END_IF;
	    END_REGION

	    REGION 8.4 - Step time watchdog
	        // the function is too long active
	        IF #iqx_Enable AND "DB_Memory"."OS_0.1sec"
	        THEN
	            #si_StepTime += 1;
	        END_IF;
	        IF (#si_StepTime > #ci_MaxStepTime)
	        THEN
	            #sa_Status.TimeExceeded := TRUE;
	        ELSE
	            #sa_Status.TimeExceeded := FALSE;
	        END_IF;
	    END_REGION
	END_REGION

	REGION 9 - Go to next step

	    IF #iqx_Enable
	        AND #sa_Status.StepDone
	        AND "DB_Memory".OS_2sec
	    THEN
	        #sx_PreparedData := FALSE;
	        #sa_Status.StepDone := FALSE;
	        #sa_Status.StepNr += 1;
	        #si_StepTime := 0;
	    END_IF;
	END_REGION

	REGION 10 - Commissioning done

	    IF (#si_StepMax <= #sa_Status.StepNr
	        AND #iqx_Enable)
	    THEN
	        #iqx_Enable := FALSE;
	        #sx_Done := TRUE;
	        #sx_Start := FALSE;
	        #sx_Busy := FALSE;
	        #sx_24VCommissioningDone := TRUE;

	    END_IF;
	END_REGION

	REGION 11 - Write output

	    #qx_Busy := #sx_Busy;
	    #qx_Done := #sx_Done;
	    #qx_Error := #sx_Error;
	    #qx_24VCommissioningDone := #sx_24VCommissioningDone;

	END_REGION


END_FUNCTION_BLOCK

TYPE "UDT_CaljanSend"
VERSION : 0.1
   STRUCT
      PEC_Override { ExternalAccessible := 'False'; ExternalVisible := 'False'; ExternalWritable := 'False'} : Bool;   // True if passage of parcels through PEC is allowed. (HMI)
      AllowLoading { ExternalAccessible := 'False'; ExternalVisible := 'False'; ExternalWritable := 'False'} : Bool;   // True if belt start in loading mode is allowed
      AllowUnloading { ExternalAccessible := 'False'; ExternalVisible := 'False'; ExternalWritable := 'False'} : Bool;   // True if belt start in unloading mode is allowed
      Reset { ExternalAccessible := 'False'; ExternalVisible := 'False'; ExternalWritable := 'False'} : Bool;   // Reset error and safety command
      "Spare_Q0.4" { ExternalAccessible := 'False'; ExternalVisible := 'False'; ExternalWritable := 'False'} : Bool;   // Spare Bit 4
      "Spare_Q0.5" : Bool := FALSE;   // Spare Bit 5
      "Spare_Q0.6" : Bool := FALSE;   // Spare Bit 6
      "Spare_Q0.7" : Bool := FALSE;   // Spare Bit 7
      Spare_QB1 : Byte;   // Spare Byte 1
      Spare_QW2 : Word;   // Spare Word 2
      Spare_QW4 : Word := 16#0000;   // Spare Word 4
      Spare_QW6 : Word := 16#0000;   // Spare Word 6
   END_STRUCT;

END_TYPE

TYPE "UDT_CaljanStatus"
TITLE = UDT_UnloaderStatus
VERSION : 0.1
//User-defined structure of FB_Unloader function block status.
   STRUCT
      Status : Int;   // Status number
      Specific : Struct   // Equipment specific warnings and errors
         PEC_EoS : "UDT_PECStatus";   // PEC status structure
         PNSlaveNotOnline { ExternalAccessible := 'False'; ExternalVisible := 'False'; ExternalWritable := 'False'} : Bool;   // Profinet slave is not online
         PNSlaveError { ExternalAccessible := 'False'; ExternalVisible := 'False'; ExternalWritable := 'False'} : Bool;   // Profinet slave is in error
         PNSlaveWarning { ExternalAccessible := 'False'; ExternalVisible := 'False'; ExternalWritable := 'False'} : Bool;   // Profinet slave has  a warning
         Disabled { ExternalAccessible := 'False'; ExternalVisible := 'False'; ExternalWritable := 'False'} : Bool;   // Unloader is disabled by HMI
         TooLongParcel { ExternalAccessible := 'False'; ExternalVisible := 'False'; ExternalWritable := 'False'} : Bool;   // Unloader detected a too long parcel
         VFDError { ExternalAccessible := 'False'; ExternalVisible := 'False'; ExternalWritable := 'False'} : Bool;   // Unloader has an VFD error
         NotHealthy { ExternalAccessible := 'False'; ExternalVisible := 'False'; ExternalWritable := 'False'} : Bool;   // Unloader is not healthy
      END_STRUCT;
   END_STRUCT;

END_TYPE

TYPE "UDT_AixZpaFullIN"
VERSION : 0.1
   STRUCT
      LocalUpstreamZoneStatus_Rev { ExternalVisible := 'False'} : Byte;   // Local upstream Zone's status when the conveyor is running in opposite to configured direction
      LocalUpstreamZoneStatus_Fwd { ExternalVisible := 'False'} : Byte;   // Local upstream Zone's status when the conveyor is running in configured direction
      LocalDownstreamZoneStatus_Rev { ExternalVisible := 'False'} : Byte;   // Local downstream Zone's status when the conveyor is running in opposite to configured direction
      LocalDownstreamZoneStatus_Fwd { ExternalVisible := 'False'} : Byte;   // Local downstream Zone's status when the conveyor is running in configured direction
      ArrivalCountUpstreamZone { ExternalVisible := 'False'} : Int;   // Count incremented upon each new arrival
      DepartureCountUpstreamZone { ExternalVisible := 'False'} : Int;   // Count incremented upon each release
      ArrivalCountDownstreamZone { ExternalVisible := 'False'} : Int;   // Count incremented upon each new arrival
      DepartureCountDownstreamZone { ExternalVisible := 'False'} : Int;   // Count incremented upon each release
      Diagnostic { ExternalVisible := 'False'} : Struct   // 32 bit diagnostic field. When bits are set the error is active
         LeftMotorOverheat { ExternalAccessible := 'False'; ExternalVisible := 'False'; ExternalWritable := 'False'} : Bool;   // Left motor temperature has exceeded 105 degrees Celsius
         LeftMotorMaxTorque { ExternalAccessible := 'False'; ExternalVisible := 'False'; ExternalWritable := 'False'} : Bool;   // Left motor is running with maximum torque output
         LeftMotorShort { ExternalAccessible := 'False'; ExternalVisible := 'False'; ExternalWritable := 'False'} : Bool;   // Left motor short circuit
         LeftMotorNotConn { ExternalAccessible := 'False'; ExternalVisible := 'False'; ExternalWritable := 'False'} : Bool;   // Left motor is not connected
         LeftMotorOverload { ExternalAccessible := 'False'; ExternalVisible := 'False'; ExternalWritable := 'False'} : Bool;   // Left motor overloaded after more than 20 seconds in Stalled
         LeftMotorStalled { ExternalAccessible := 'False'; ExternalVisible := 'False'; ExternalWritable := 'False'} : Bool;   // Left motor stalled and speed is less than 10% of the set speed
         LeftMotorBadHall { ExternalAccessible := 'False'; ExternalVisible := 'False'; ExternalWritable := 'False'} : Bool;   // Left motor Hall Efect Sensor error active
         LeftMotorNotUsed { ExternalAccessible := 'False'; ExternalVisible := 'False'; ExternalWritable := 'False'} : Bool;   // Left motor is not used
         ModuleResetFlag { ExternalAccessible := 'False'; ExternalVisible := 'False'; ExternalWritable := 'False'} : Bool;
         Index06Bit01 { ExternalAccessible := 'False'; ExternalVisible := 'False'; ExternalWritable := 'False'} : Bool;   // Reserved
         OverVoltage { ExternalAccessible := 'False'; ExternalVisible := 'False'; ExternalWritable := 'False'} : Bool;   // Supply voltage + Left motor back EMF exceeded 30 volts
         LeftMotorAnyErr { ExternalAccessible := 'False'; ExternalVisible := 'False'; ExternalWritable := 'False'} : Bool;   // Any Left motor error active
         ConnectionsNotOK { ExternalAccessible := 'False'; ExternalVisible := 'False'; ExternalWritable := 'False'} : Bool;   // Ethernet connection error
         UpstreamJamErr { ExternalAccessible := 'False'; ExternalVisible := 'False'; ExternalWritable := 'False'} : Bool;   // Jam error active on Upstream zone
         LeftSensLowGain { ExternalAccessible := 'False'; ExternalVisible := 'False'; ExternalWritable := 'False'} : Bool;   // Left sensor error
         LowVoltage { ExternalAccessible := 'False'; ExternalVisible := 'False'; ExternalWritable := 'False'} : Bool;   // Module power supply is less than 18 Volts
         RightMotorOverheat { ExternalAccessible := 'False'; ExternalVisible := 'False'; ExternalWritable := 'False'} : Bool;   // Right motor temperature has exceeded 105 degrees Celsius
         RightMotorMaxTorque { ExternalAccessible := 'False'; ExternalVisible := 'False'; ExternalWritable := 'False'} : Bool;   // Right motor is running with maximum torque output
         RightMotorShort { ExternalAccessible := 'False'; ExternalVisible := 'False'; ExternalWritable := 'False'} : Bool;   // Right motor short circuit
         RightMotorNotConn { ExternalAccessible := 'False'; ExternalVisible := 'False'; ExternalWritable := 'False'} : Bool;   // Right motor is not connected
         RightMotorOverload { ExternalAccessible := 'False'; ExternalVisible := 'False'; ExternalWritable := 'False'} : Bool;   // Right motor overloaded after more than 20 seconds in Stalled
         RightMotorStalled { ExternalAccessible := 'False'; ExternalVisible := 'False'; ExternalWritable := 'False'} : Bool;   // Right motor is stalled and speed is less than 10% of the set speed
         RightMotorBadHall { ExternalAccessible := 'False'; ExternalVisible := 'False'; ExternalWritable := 'False'} : Bool;   // Right motor Hall Efect Sensor error active
         RightMotorNotUsed { ExternalAccessible := 'False'; ExternalVisible := 'False'; ExternalWritable := 'False'} : Bool;   // Right motor is not used
         Index07Bit00 { ExternalAccessible := 'False'; ExternalVisible := 'False'; ExternalWritable := 'False'} : Bool;   // Reserved
         Index07Bit01 { ExternalAccessible := 'False'; ExternalVisible := 'False'; ExternalWritable := 'False'} : Bool;   // Reserved
         OverVoltage1 { ExternalAccessible := 'False'; ExternalVisible := 'False'; ExternalWritable := 'False'} : Bool;   // Supply voltage + Right motor back EMF exceeded 30 volts
         RightMotorAnyErr { ExternalAccessible := 'False'; ExternalVisible := 'False'; ExternalWritable := 'False'} : Bool;   // Any Right motor error active
         Index07Bit04 { ExternalAccessible := 'False'; ExternalVisible := 'False'; ExternalWritable := 'False'} : Bool;   // Reserved
         DownstreamJamErr { ExternalAccessible := 'False'; ExternalVisible := 'False'; ExternalWritable := 'False'} : Bool;   // Jam error active on Downstream zone
         RightSensLowGain { ExternalAccessible := 'False'; ExternalVisible := 'False'; ExternalWritable := 'False'} : Bool;   // Right sensor error
         LowVoltage1 { ExternalAccessible := 'False'; ExternalVisible := 'False'; ExternalWritable := 'False'} : Bool;   // Module power supply is less than 18 Volts
      END_STRUCT;
      TrackingUpstreamZone { ExternalVisible := 'False'} : DWord;   // The Tracking data of the product currently on this zone
      TrackingDownstreamZone { ExternalVisible := 'False'} : DWord;   // The Tracking data of the product currently on this zone
      ReleaseCounterUpstreamZone { ExternalVisible := 'False'} : Int;   // Current value of the 'SetReleaseCountUpstream' output
      ReleaseCounterDownstreamZone { ExternalVisible := 'False'} : Int;   // Current value of the 'SetReleaseCountDownstream' output
      GetDischargeTracking_Fwd { ExternalVisible := 'False'} : DWord;   // Tracking data of just discharged item when running in configured direction
      GetDischargeTracking_Rev { ExternalVisible := 'False'} : DWord;   // Tracking data of just discharged item when running in opposite of configured direction
      AllSensorPortInputs { ExternalVisible := 'False'} : Struct   // Left and Right Sensor Port inputs
         Bit08 { ExternalAccessible := 'False'; ExternalVisible := 'False'; ExternalWritable := 'False'} : Bool;   // Reserved
         Bit09 { ExternalAccessible := 'False'; ExternalVisible := 'False'; ExternalWritable := 'False'} : Bool;   // Reserved
         Bit10 { ExternalAccessible := 'False'; ExternalVisible := 'False'; ExternalWritable := 'False'} : Bool;   // Reserved
         Bit11 { ExternalAccessible := 'False'; ExternalVisible := 'False'; ExternalWritable := 'False'} : Bool;   // Reserved
         Bit12 { ExternalAccessible := 'False'; ExternalVisible := 'False'; ExternalWritable := 'False'} : Bool;   // Reserved
         Bit13 { ExternalAccessible := 'False'; ExternalVisible := 'False'; ExternalWritable := 'False'} : Bool;   // Reserved
         Bit14 { ExternalAccessible := 'False'; ExternalVisible := 'False'; ExternalWritable := 'False'} : Bool;   // Reserved
         Heartbeat { ExternalAccessible := 'False'; ExternalVisible := 'False'; ExternalWritable := 'False'} : Bool;   // This bit toggles every 2 seconds
         LeftPin2 { ExternalAccessible := 'False'; ExternalVisible := 'False'; ExternalWritable := 'False'} : Bool;   // Left sensor port state (Pin2)
         Bit01 { ExternalAccessible := 'False'; ExternalVisible := 'False'; ExternalWritable := 'False'} : Bool;   // Reserved
         RightPin2 { ExternalAccessible := 'False'; ExternalVisible := 'False'; ExternalWritable := 'False'} : Bool;   // Right sensor port state (Pin2)
         Bit03 { ExternalAccessible := 'False'; ExternalVisible := 'False'; ExternalWritable := 'False'} : Bool;   // Reserved
         LeftSensor { ExternalAccessible := 'False'; ExternalVisible := 'False'; ExternalWritable := 'False'} : Bool;   // Left sensor port state (Pin4)
         Bit05 { ExternalAccessible := 'False'; ExternalVisible := 'False'; ExternalWritable := 'False'} : Bool;   // Reserved
         RightSensor { ExternalAccessible := 'False'; ExternalVisible := 'False'; ExternalWritable := 'False'} : Bool;   // Right sensor port state (Pin4)
         Bit07 { ExternalAccessible := 'False'; ExternalVisible := 'False'; ExternalWritable := 'False'} : Bool;   // Reserved
      END_STRUCT;
      Index19 { ExternalVisible := 'False'} : Word;   // Reserved
      ConveyStopStatus { ExternalVisible := 'False'} : Struct   // Status of ConveyStop
         Bit08 { ExternalAccessible := 'False'; ExternalVisible := 'False'; ExternalWritable := 'False'} : Bool;   // Reserved
         Bit09 { ExternalAccessible := 'False'; ExternalVisible := 'False'; ExternalWritable := 'False'} : Bool;   // Reserved
         StopActiveCommandPLC { ExternalAccessible := 'False'; ExternalVisible := 'False'; ExternalWritable := 'False'} : Bool;   // Stop active due to stop command from the PLC
         Bit11 { ExternalAccessible := 'False'; ExternalVisible := 'False'; ExternalWritable := 'False'} : Bool;   // Reserved
         Bit12 { ExternalAccessible := 'False'; ExternalVisible := 'False'; ExternalWritable := 'False'} : Bool;   // Reserved
         Bit13 { ExternalAccessible := 'False'; ExternalVisible := 'False'; ExternalWritable := 'False'} : Bool;   // Reserved
         Bit14 { ExternalAccessible := 'False'; ExternalVisible := 'False'; ExternalWritable := 'False'} : Bool;   // Reserved
         Bit15 { ExternalAccessible := 'False'; ExternalVisible := 'False'; ExternalWritable := 'False'} : Bool;   // Reserved
         Bit00 { ExternalAccessible := 'False'; ExternalVisible := 'False'; ExternalWritable := 'False'} : Bool;   // Reserved
         Bit01 { ExternalAccessible := 'False'; ExternalVisible := 'False'; ExternalWritable := 'False'} : Bool;   // Reserved
         Bit02 { ExternalAccessible := 'False'; ExternalVisible := 'False'; ExternalWritable := 'False'} : Bool;   // Reserved
         Bit03 { ExternalAccessible := 'False'; ExternalVisible := 'False'; ExternalWritable := 'False'} : Bool;   // Reserved
         Bit04 { ExternalAccessible := 'False'; ExternalVisible := 'False'; ExternalWritable := 'False'} : Bool;   // Reserved
         StopActiveOtherModule { ExternalAccessible := 'False'; ExternalVisible := 'False'; ExternalWritable := 'False'} : Bool;   // Stop condition is active on a module in the ConveyStop group
         StopActiveLostConn { ExternalAccessible := 'False'; ExternalVisible := 'False'; ExternalWritable := 'False'} : Bool;   // Stop is active due to a loss of communication connection
         StopActiveLostPLC { ExternalAccessible := 'False'; ExternalVisible := 'False'; ExternalWritable := 'False'} : Bool;   // Stop active due to a loss of connection with the PLC
      END_STRUCT;
      Future { ExternalVisible := 'False'} : Array[21..30] of Int;
      GeneralLineError : Struct
         Reserved0 { ExternalAccessible := 'False'; ExternalVisible := 'False'; ExternalWritable := 'False'} : Bool;
         Reserved1 { ExternalAccessible := 'False'; ExternalVisible := 'False'; ExternalWritable := 'False'} : Bool;
         Reserved2 { ExternalAccessible := 'False'; ExternalVisible := 'False'; ExternalWritable := 'False'} : Bool;
         Reserved3 { ExternalAccessible := 'False'; ExternalVisible := 'False'; ExternalWritable := 'False'} : Bool;
         Reserved4 { ExternalAccessible := 'False'; ExternalVisible := 'False'; ExternalWritable := 'False'} : Bool;
         Reserved5 { ExternalAccessible := 'False'; ExternalVisible := 'False'; ExternalWritable := 'False'} : Bool;
         Reserved6 { ExternalAccessible := 'False'; ExternalVisible := 'False'; ExternalWritable := 'False'} : Bool;
         Reserved7 { ExternalAccessible := 'False'; ExternalVisible := 'False'; ExternalWritable := 'False'} : Bool;
         MotorError { ExternalAccessible := 'False'; ExternalVisible := 'False'; ExternalWritable := 'False'} : Bool;   // There is a motor error somewhere upstream
         ConnectionError { ExternalAccessible := 'False'; ExternalVisible := 'False'; ExternalWritable := 'False'} : Bool;   // There is a connection error somewhere upstream
         JamError { ExternalAccessible := 'False'; ExternalVisible := 'False'; ExternalWritable := 'False'} : Bool;   // There is a Jam error somewhere upstream
         SensorDetectError { ExternalAccessible := 'False'; ExternalVisible := 'False'; ExternalWritable := 'False'} : Bool;   // There is a Sensor detect error somewhere upstream
         Reserved12 { ExternalAccessible := 'False'; ExternalVisible := 'False'; ExternalWritable := 'False'} : Bool;
         Reserved13 { ExternalAccessible := 'False'; ExternalVisible := 'False'; ExternalWritable := 'False'} : Bool;
         Reserved14 { ExternalAccessible := 'False'; ExternalVisible := 'False'; ExternalWritable := 'False'} : Bool;
         Reserved15 { ExternalAccessible := 'False'; ExternalVisible := 'False'; ExternalWritable := 'False'} : Bool;
      END_STRUCT;
   END_STRUCT;

END_TYPE

TYPE "UDT_CaljanReceive"
VERSION : 0.1
   STRUCT
      Healthy { ExternalAccessible := 'False'; ExternalVisible := 'False'; ExternalWritable := 'False'} : Bool;   // True if (un)loader is healthy
      BeltDirection_Loading { ExternalAccessible := 'False'; ExternalVisible := 'False'; ExternalWritable := 'False'} : Bool;   // True if belt is running in loading mode
      BeltDirection_Unloading { ExternalAccessible := 'False'; ExternalVisible := 'False'; ExternalWritable := 'False'} : Bool;   // True if belt is running in unloading mode
      ReadyToReceive { ExternalAccessible := 'False'; ExternalVisible := 'False'; ExternalWritable := 'False'} : Bool;   // True if loader is ready to receive
      HoldReverseSignal { ExternalAccessible := 'False'; ExternalVisible := 'False'; ExternalWritable := 'False'} : Bool;   // True when reverse button is pressed (only applicable to unloaders)
      ResetReverse { ExternalAccessible := 'False'; ExternalVisible := 'False'; ExternalWritable := 'False'} : Bool;   // True when reset reverse button is pressed (only applicable to unloaders)
      PECUnloader { ExternalAccessible := 'False'; ExternalVisible := 'False'; ExternalWritable := 'False'} : Bool;   // True when no parcels are detected (fail safe)
      "Spare_I0.7" { ExternalAccessible := 'False'; ExternalVisible := 'False'; ExternalWritable := 'False'} : Bool;   // Spare Bit 7
      Spare_IB1 : Byte;   // Spare Byte 1
      ActualSpeed : Int;   // Actual speed [mm/s]
      Spare_IW4 : Word;   // Spare Word 3
      Spare_IW6 : Word;   // Spare Word 4
   END_STRUCT;

END_TYPE

TYPE "UDT_AixZpaFullOUT"
VERSION : 0.1
   STRUCT
      InductTrackingOnUpstreamZone { ExternalVisible := 'False'} : DWord;   // Writes the tracking data of the product currently on the zone when ReleaseControlUpstream is incremented by 1
      InductTrackingOnDownstreamZone { ExternalVisible := 'False'} : DWord;   // Writes the tracking data of the product currently on the zone when ReleaseControlDownstream is incremented by 1
      AccumulateControlUpstream { ExternalVisible := 'False'} : Struct
         AccumUpstreamToThisZone { ExternalAccessible := 'False'; ExternalVisible := 'False'; ExternalWritable := 'False'} : Bool;   // Accumulates the Upstream zone relative to this zone
         SetArrival { ExternalAccessible := 'False'; ExternalVisible := 'False'; ExternalWritable := 'False'} : Bool;   // Simulate downstream arrival to prevent Arrival Jam
         JogDefaultDir { ExternalAccessible := 'False'; ExternalVisible := 'False'; ExternalWritable := 'False'} : Bool;   // Jog zone in default direction
         JogOppDir { ExternalAccessible := 'False'; ExternalVisible := 'False'; ExternalWritable := 'False'} : Bool;   // Jog zone in opposite of default direction
         WakeUp { ExternalAccessible := 'False'; ExternalVisible := 'False'; ExternalWritable := 'False'} : Bool;   // Wake Up Local Upstream Zone
         MaintMode { ExternalAccessible := 'False'; ExternalVisible := 'False'; ExternalWritable := 'False'} : Bool;   // Enable Maintenance Mode
         Bit14 { ExternalAccessible := 'False'; ExternalVisible := 'False'; ExternalWritable := 'False'} : Bool;   // Reserved
         Bit15 { ExternalAccessible := 'False'; ExternalVisible := 'False'; ExternalWritable := 'False'} : Bool;   // Reserved
         Accumulate { ExternalAccessible := 'False'; ExternalVisible := 'False'; ExternalWritable := 'False'} : Bool;   // Accumulates this local zone
         Bit01 { ExternalAccessible := 'False'; ExternalVisible := 'False'; ExternalWritable := 'False'} : Bool;   // Reserved
         Bit02 { ExternalAccessible := 'False'; ExternalVisible := 'False'; ExternalWritable := 'False'} : Bool;   // Reserved
         Bit03 { ExternalAccessible := 'False'; ExternalVisible := 'False'; ExternalWritable := 'False'} : Bool;   // Reserved
         Bit04 { ExternalAccessible := 'False'; ExternalVisible := 'False'; ExternalWritable := 'False'} : Bool;   // Reserved
         Bit05 { ExternalAccessible := 'False'; ExternalVisible := 'False'; ExternalWritable := 'False'} : Bool;   // Reserved
         Bit06 { ExternalAccessible := 'False'; ExternalVisible := 'False'; ExternalWritable := 'False'} : Bool;   // Reserved
         Bit07 { ExternalAccessible := 'False'; ExternalVisible := 'False'; ExternalWritable := 'False'} : Bool;   // Reserved
      END_STRUCT;
      AccumulateControlDownstream { ExternalVisible := 'False'} : Struct
         AccumUpstreamToThisZone { ExternalAccessible := 'False'; ExternalVisible := 'False'; ExternalWritable := 'False'} : Bool;   // Accumulates the Upstream zone relative to this zone
         SetArrival { ExternalAccessible := 'False'; ExternalVisible := 'False'; ExternalWritable := 'False'} : Bool;   // Simulate downstream arrival to prevent Arrival Jam
         JogDefaultDir { ExternalAccessible := 'False'; ExternalVisible := 'False'; ExternalWritable := 'False'} : Bool;   // Jog zone in default direction
         JogOppDir { ExternalAccessible := 'False'; ExternalVisible := 'False'; ExternalWritable := 'False'} : Bool;   // Jog zone in opposite of default direction
         WakeUp { ExternalAccessible := 'False'; ExternalVisible := 'False'; ExternalWritable := 'False'} : Bool;   // Wake Up Local Downstream Zone
         MaintMode { ExternalAccessible := 'False'; ExternalVisible := 'False'; ExternalWritable := 'False'} : Bool;   // Enable Maintenance Moded
         Bit14 { ExternalAccessible := 'False'; ExternalVisible := 'False'; ExternalWritable := 'False'} : Bool;   // Reserved
         Bit15 { ExternalAccessible := 'False'; ExternalVisible := 'False'; ExternalWritable := 'False'} : Bool;   // Reserved
         Accumulate { ExternalAccessible := 'False'; ExternalVisible := 'False'; ExternalWritable := 'False'} : Bool;   // Accumulates this local zone
         Bit01 { ExternalAccessible := 'False'; ExternalVisible := 'False'; ExternalWritable := 'False'} : Bool;   // Reserved
         Bit02 { ExternalAccessible := 'False'; ExternalVisible := 'False'; ExternalWritable := 'False'} : Bool;   // Reserved
         Bit03 { ExternalAccessible := 'False'; ExternalVisible := 'False'; ExternalWritable := 'False'} : Bool;   // Reserved
         Bit04 { ExternalAccessible := 'False'; ExternalVisible := 'False'; ExternalWritable := 'False'} : Bool;   // Reserved
         Bit05 { ExternalAccessible := 'False'; ExternalVisible := 'False'; ExternalWritable := 'False'} : Bool;   // Reserved
         Bit06 { ExternalAccessible := 'False'; ExternalVisible := 'False'; ExternalWritable := 'False'} : Bool;   // Reserved
         Bit07 { ExternalAccessible := 'False'; ExternalVisible := 'False'; ExternalWritable := 'False'} : Bool;   // Reserved
      END_STRUCT;
      SetSpeedLeftMotor { ExternalVisible := 'False'} : Int;   // Speed setting for Left motor in mm/s(or 1/10 of an RPM for PGD)
      SetSpeedRightMotor { ExternalVisible := 'False'} : Int;   // Speed setting for the Right motor in mm/s(or 1/10 of an RPM for PGD)
      SetReleaseCountUpstream { ExternalVisible := 'False'} : Int;   // Changing the value causes the Upstream zone to release the current product
      SetReleaseCountDownstream { ExternalVisible := 'False'} : Int;   // Changing the value causes the Downstream zone to release the current product
      SetInductStatus { ExternalVisible := 'False'} : Word;   // Used as a "Wake up" signal - Write '4' to wake up, write 1 to stop wake up
      SetDishargeStatus { ExternalVisible := 'False'} : Word;   // Used as a "Lane full" signal. Write '5' to accumulate, write 1 to allow release
      SetInductTrackingFwd { ExternalVisible := 'False'} : DWord;   // Assign this data to next arrival when in fwd direction
      SetInductTrackingRev { ExternalVisible := 'False'} : DWord;   // Assign this data to next arrival when in rev direction
      ClearMotorError { ExternalVisible := 'False'} : Word;   // Write '1" to clear motor error - Write '0' to resume
      Index17 { ExternalVisible := 'False'} : Word;   // Reserved
      Index18 { ExternalVisible := 'False'} : Word;   // Reserved
      ConveyStopControl { ExternalVisible := 'False'} : Word;   // Write '1' to STOP the group, write 2 to clear STOP. Transition 0 - 2 is needed to clear the Stop
      ClearJamUpstream { ExternalVisible := 'False'} : Word;   // Write '1' to clear zone jam
      ClearJamDownstream { ExternalVisible := 'False'} : Word;   // Write '1' to clear zone jam
      GlobalDirAccModeUpstr { ExternalVisible := 'False'} : Word;   // Used to change direction of flow or accumulation mode for a continuous group of zones beginning with the local zone
      GlobalDirAccModeDnstr { ExternalVisible := 'False'} : Word;   // Used to change direction of flow or accumulation mode for a continuous group of zones beginning with the local zone
      Future { ExternalVisible := 'False'} : Array[24..31] of Int;
   END_STRUCT;

END_TYPE

TYPE "UDT_ConveyorStatus"
TITLE = UDT_ConveyorStatus
VERSION : 0.1
//User-defined structure of FB_Conveyor function block status.
   STRUCT
      Status : Int;   // Status number
      Specific : Struct
         Reverse { ExternalAccessible := 'False'; ExternalVisible := 'False'; ExternalWritable := 'False'} : Bool;   // Conveyor is running in reverse direction
      END_STRUCT;
   END_STRUCT;

END_TYPE

TYPE "UDT_CaljanConfiguration"
TITLE = UDT_UnloaderConfiguration
VERSION : 0.1
//User-defined structure of unloader parameters.
   STRUCT
      PEC_EOS : "UDT_PECConfiguration";   // Photo eye time on delay
      Forward_Direction : Struct   // Forward Direction configuration
         GapHeadToHead : DInt;   // Gapping head to head value [cm]
         GapTailToHead : DInt;   // Gapping tail to head value [cm]
         GapCorrection : DInt;   // Gap offset to cover VFD's ramps [cm]
      END_STRUCT;
      PNDeviceName : String;   // VFD's Profinet device name
      Speedsetpoint : Int;   // Speedsetpoint: 0=Low, 1=Nom, 2=High
      EnergySaveLength : Int;   // Distance conveyor traveled before energy save activate [cm]
      FirstConveyorToStart { ExternalAccessible := 'False'; ExternalVisible := 'False'; ExternalWritable := 'False'} : Bool;   // First conveyor to start cascade mode
      Energy { ExternalAccessible := 'False'; ExternalVisible := 'False'; ExternalWritable := 'False'} : Bool;   // Energy save mode enable
      ResetDelay : UDInt := 1000;   // Time required
      CaljanMode : Int;   // Choosing device 1=loader, 2=unloader
      CascadeTimeOnDelay : UDInt;   // Cascade time on delay [ms]
   END_STRUCT;

END_TYPE

TYPE "UDT_ConveyorCommand"
TITLE = UDT_ConveyorCommand
VERSION : 0.1
//User-defined structure of conveyor commands.
   STRUCT
      ManualMode { ExternalAccessible := 'False'; ExternalVisible := 'False'; ExternalWritable := 'False'} : Bool;   // Manual mode command from HMI
      ManualStartStop { ExternalAccessible := 'False'; ExternalVisible := 'False'; ExternalWritable := 'False'} : Bool;   // Run conveyor in manual mode
      ManualFullSpeed { ExternalAccessible := 'False'; ExternalVisible := 'False'; ExternalWritable := 'False'} : Bool;   // Full speed conveyor in manual mode
      ManualJog { ExternalAccessible := 'False'; ExternalVisible := 'False'; ExternalWritable := 'False'} : Bool;   // Command to jog conveyor in slow speed from HMI
      Reverse { ExternalAccessible := 'False'; ExternalVisible := 'False'; ExternalWritable := 'False'} : Bool;   // Command to run conveyor in reverse direction from HMI
      ManualSpeed : Int := 50;   // Manual mode speed as percentage of nominal speed [0-100%]
   END_STRUCT;

END_TYPE

TYPE "UDT_Interface_Signal"
VERSION : 0.1
   STRUCT
      RQST { ExternalAccessible := 'False'; ExternalVisible := 'False'; ExternalWritable := 'False'} : Bool;   // Request to activate
      CMD { ExternalAccessible := 'False'; ExternalVisible := 'False'; ExternalWritable := 'False'} : Bool;   // Request is Active and thus commanded
   END_STRUCT;

END_TYPE

TYPE "UDT_UnloaderStatus"
TITLE = UDT_UnloaderStatus
VERSION : 0.1
//User-defined structure of FB_Unloader function block status.
   STRUCT
      Status : Int;   // Status number
      Specific : Struct   // Equipment specific warnings and errors
         PEC_EoS : "UDT_PECStatus";   // PEC status structure
         Disabled { ExternalAccessible := 'False'; ExternalVisible := 'False'; ExternalWritable := 'False'} : Bool;   // Unloader is disabled by HMI
         TooLongParcel { ExternalAccessible := 'False'; ExternalVisible := 'False'; ExternalWritable := 'False'} : Bool;   // Unloader detected a too long parcel
         VFDError { ExternalAccessible := 'False'; ExternalVisible := 'False'; ExternalWritable := 'False'} : Bool;   // Unloader has an VFD error
         NotHealthy { ExternalAccessible := 'False'; ExternalVisible := 'False'; ExternalWritable := 'False'} : Bool;   // Unloader is not healthy
      END_STRUCT;
   END_STRUCT;

END_TYPE

TYPE "UDT_PNNodeStatus"
VERSION : 0.1
   STRUCT
      Status : Int;   // Status number
      Specific : Struct   // Specific structure
         PNSlaveNotOnline { ExternalAccessible := 'False'; ExternalVisible := 'False'; ExternalWritable := 'False'} : Bool;   // Profinet slave is not online
         PNSlaveError { ExternalAccessible := 'False'; ExternalVisible := 'False'; ExternalWritable := 'False'} : Bool;   // Profinet slave is in error
         PNSlaveWarning { ExternalAccessible := 'False'; ExternalVisible := 'False'; ExternalWritable := 'False'} : Bool;   // Profinet slave has  a warning
      END_STRUCT;
   END_STRUCT;

END_TYPE

FUNCTION_BLOCK "FB_AMBASpiralChainCheck"
{ S7_Optimized_Access := 'TRUE' }
VERSION : 0.1
// ATTRIBUTES
// AUTO_NUMBER = True
// BLOCK_NUMBER = 256
// END_ATTRIBUTES
   VAR_INPUT
      ix_ProxSwitchDriveShaft { ExternalAccessible := 'False'; ExternalVisible := 'False'; ExternalWritable := 'False'} : Bool;   // Proximity switche signal drive shaft
      ix_ProxSwitchIdlerShaft { ExternalAccessible := 'False'; ExternalVisible := 'False'; ExternalWritable := 'False'} : Bool;   // Proximity switche signal idler shaft
      ix_HardwareOK { ExternalAccessible := 'False'; ExternalVisible := 'False'; ExternalWritable := 'False'} : Bool;   // TRUE when hardware is ok
   END_VAR

   VAR_IN_OUT
      iqx_BrokenChainDetected { ExternalAccessible := 'False'; ExternalVisible := 'False'; ExternalWritable := 'False'} : Bool;   // [Failure] Broken chain detected (TRUE = detected)
      iqx_ChainOverlengthDetected { ExternalAccessible := 'False'; ExternalVisible := 'False'; ExternalWritable := 'False'} : Bool;   // [Warning] Chain overlength detected (TRUE = detected)
      iqUDT_BrokenChainStatistics : "UDT_EventStatistic";   // Statistics of broken chain event
      iqUDT_ChainOverlengthStatistics : "UDT_EventStatistic";   // Statistics of missing slat event
      iqUDT_EquipmentControl : "UDT_EquipmentControl";
   END_VAR

   VAR
      sFB_SignalFilter_DriveShaft { ExternalAccessible := 'False'; ExternalVisible := 'False'; ExternalWritable := 'False'; S7_SetPoint := 'False'} : "FB_TimerOnOffDelay";   // On/Off delay to filter the input signal
      sFB_SignalFilter_IdlerShaft { ExternalAccessible := 'False'; ExternalVisible := 'False'; ExternalWritable := 'False'; S7_SetPoint := 'False'} : "FB_TimerOnOffDelay";   // On/Off delay to filter the input signal
      sR_TRIG_DriveShaft {InstructionName := 'R_TRIG'; LibVersion := '1.0'; ExternalAccessible := 'False'; ExternalVisible := 'False'; ExternalWritable := 'False'; S7_SetPoint := 'False'} : R_TRIG;
      sR_TRIG_IdlerShaft {InstructionName := 'R_TRIG'; LibVersion := '1.0'; ExternalAccessible := 'False'; ExternalVisible := 'False'; ExternalWritable := 'False'; S7_SetPoint := 'False'} : R_TRIG;
      sR_TRIG_ChainOverlength {InstructionName := 'R_TRIG'; LibVersion := '1.0'; ExternalAccessible := 'False'; ExternalVisible := 'False'; ExternalWritable := 'False'; S7_SetPoint := 'False'} : R_TRIG;
      sR_TRIG_BrokenChain {InstructionName := 'R_TRIG'; LibVersion := '1.0'; ExternalAccessible := 'False'; ExternalVisible := 'False'; ExternalWritable := 'False'; S7_SetPoint := 'False'} : R_TRIG;
      si_PulseCounterDriveShaft { ExternalAccessible := 'False'; ExternalVisible := 'False'; ExternalWritable := 'False'} : Int;   // Counter drive shaft pulses
      sx_IdlerShaftPulse { ExternalAccessible := 'False'; ExternalVisible := 'False'; ExternalWritable := 'False'} : Bool;
   END_VAR

   VAR CONSTANT
      cudi_OffDelay : UDInt := 25;   // [ms]
      cudi_OnDelay : UDInt := 25;   // [ms]
   END_VAR


BEGIN
	(*
	Version history:
	Date        | Version   | Author              | Remark
	----------------------------------------------------------------------------------------
	 14/03/2022 | 1.0       | G.Vlooswijk         | Initial version for FedEx Milano
	 16/05/2022 | 1.1       | G.Vlooswijk         | Tested (logic) GLS Tongeren
	 03/06/2024 | 1.2       | J.Majer             | Adapted to current library
	*)

	REGION Input signals

	    //Filter signals
	    #sFB_SignalFilter_DriveShaft(iudi_OnDelayTime := #cudi_OnDelay,
	                                 iudi_OffDelayTime := #cudi_OffDelay,
	                                 ix_SignalToDelay := #ix_ProxSwitchDriveShaft);

	    #sFB_SignalFilter_IdlerShaft(iudi_OnDelayTime := #cudi_OnDelay,
	                                 iudi_OffDelayTime := #cudi_OffDelay,
	                                 ix_SignalToDelay := #ix_ProxSwitchIdlerShaft);

	    //Flank detection
	    #sR_TRIG_DriveShaft(CLK := #sFB_SignalFilter_DriveShaft.qx_DelayedSignal);

	    #sR_TRIG_IdlerShaft(CLK := #sFB_SignalFilter_IdlerShaft.qx_DelayedSignal);

	END_REGION

	REGION Broken chain logic

	    IF #sR_TRIG_DriveShaft.Q THEN
	        #si_PulseCounterDriveShaft += 1;
	    END_IF;

	    IF #sR_TRIG_IdlerShaft.Q THEN
	        #si_PulseCounterDriveShaft := 0;
	    END_IF;

	    //Set fault
	    IF #si_PulseCounterDriveShaft > 2 AND #ix_HardwareOK THEN
	        #iqx_BrokenChainDetected := TRUE;
	    END_IF;

	    //Reset fault
	    IF #iqx_BrokenChainDetected AND NOT #ix_HardwareOK
	        OR #iqx_BrokenChainDetected AND #iqUDT_EquipmentControl.Command.Reset
	    THEN
	        #iqx_BrokenChainDetected := FALSE;
	        #si_PulseCounterDriveShaft := 0;
	    END_IF;

	END_REGION

	(* Chain overlength is detected when the drive shaft pulse is not active during the whole Idler shaft pulse. *)
	REGION Chain overlength logic

	    //Set mememory bit on rising flank Iderler shaft pulse
	    IF #sR_TRIG_IdlerShaft.Q THEN
	        #sx_IdlerShaftPulse := TRUE;
	    END_IF;

	    //Reset memory bit when both signals are high
	    IF #sFB_SignalFilter_DriveShaft.qx_DelayedSignal
	        AND #sFB_SignalFilter_IdlerShaft.qx_DelayedSignal
	        AND #sx_IdlerShaftPulse
	    THEN
	        #sx_IdlerShaftPulse := FALSE;
	    END_IF;

	    //Set warning
	    IF #sx_IdlerShaftPulse
	        AND NOT #sFB_SignalFilter_IdlerShaft.qx_DelayedSignal
	        AND #ix_HardwareOK
	    THEN
	        #iqx_ChainOverlengthDetected := TRUE;
	    END_IF;

	    //Reset warning
	    IF #iqx_ChainOverlengthDetected
	        AND (NOT #ix_HardwareOK
	        OR #iqUDT_EquipmentControl.Command.Reset)
	    THEN
	        #iqx_ChainOverlengthDetected := FALSE;
	    END_IF;

	END_REGION

	REGION Statistics

	    REGION Broken chain

	        #sR_TRIG_BrokenChain(CLK := #iqx_BrokenChainDetected);

	        IF #iqx_BrokenChainDetected
	            OR #iqUDT_EquipmentControl.Command.ResetData
	        THEN
	            "FC_Statistics"(ix_Reset := #iqUDT_EquipmentControl.Command.ResetData,
	                            ix_Activate := #iqx_BrokenChainDetected,
	                            ix_RTrigActivate := #sR_TRIG_BrokenChain.Q,
	                            iqUDT_Statistics := #iqUDT_BrokenChainStatistics);
	        END_IF;

	    END_REGION

	    REGION Chain overlength

	        #sR_TRIG_ChainOverlength(CLK := #iqx_ChainOverlengthDetected);

	        IF #iqx_ChainOverlengthDetected
	            OR #iqUDT_EquipmentControl.Command.ResetData
	        THEN
	            "FC_Statistics"(ix_Reset := #iqUDT_EquipmentControl.Command.ResetData,
	                            ix_Activate := #iqx_ChainOverlengthDetected,
	                            ix_RTrigActivate := #sR_TRIG_ChainOverlength.Q,
	                            iqUDT_Statistics := #iqUDT_ChainOverlengthStatistics);
	        END_IF;

	    END_REGION

	END_REGION

END_FUNCTION_BLOCK

FUNCTION "FC_Fifo" : Void
TITLE = FC_Fifo
{ S7_Optimized_Access := 'TRUE' }
AUTHOR : MHSE
FAMILY : GeneralSystemFunctions
VERSION : 3.0
// ATTRIBUTES
// AUTO_NUMBER = True
// BLOCK_NUMBER = 17
// END_ATTRIBUTES
//Function for controlling FIFO register.
   VAR_INPUT
      ic_Mode : Char;   // Mode selector: "W" - Write; "R" - Read; "C" - Clear (Reset) "S" - Status
   END_VAR

   VAR_OUTPUT
      qUDT_Status : "UDT_FifoStatus";   // FIFO status structure
      qx_Error : Bool;   // Collective error output
      qx_Warning : Bool;   // Collective warning output
   END_VAR

   VAR_IN_OUT
      iqv_Data : Variant;   // Data
      iqUDT_FifoHeader : "UDT_FifoHeader";   // FIFO header
      iqv_DataBuffer : Variant;   // FIFO data buffer
   END_VAR

   VAR_TEMP
      tUDT_Status : "UDT_FifoStatus";   // Status structure
      ti_MoveBLKErrorCode : Int;   // Move_BLK_Variant function return
      tx_HeaderValid : Bool;   // Header valid
   END_VAR


BEGIN
	(*
	----------------------------------------------------------------------------------------

	Version history:
	Date        | Version   | Author        | Remark
	----------------------------------------------------------------------------------------
	24/05/2019  | 0.1       | L.Klar        | first release MHS TIA 15.1
	14/06/2019  | 0.2       | A.Nowak       | Replacement of instruction if for direct write into variable - Region 3 , 4.1 , 4.2 , 4.3 , 4.4 , 8.1  , 8.2
	17/07/2019  | 0.3       | L.Klar        | Status handling changed
	24/07/2019  | 2.0       | L.Klar        | 2.0 MHS library release TIA 15.1
	23/08/2019  | 2.1       | K.Pokorski    | Comments corrected
	27/08/2019  | 2.2       | M.Kurpiers    | Comments adjusted
	27/09/2019  | 2.3       | K.Pokorski    | Variant input included
	01/10/2019  | 2.4       | A.Nowak       | Correct comments and rename regions
	12/11/2019  | 3.0       | P.Majka       | 3.0 MHS library release TIA 15.1
	21/02/2023  | 4.0       | F.Baten       | 4.0 Release TIA 17.5
	*)

	REGION 1 – Diagnostic bits initialization

	    // Clear FIFO statuses
	    #tUDT_Status.FifoFull := FALSE;
	    #tUDT_Status.FifoPreFull := FALSE;

	END_REGION

	REGION 2 – Array's information

	    // If buffer elements type is invalid, set the error
	    #tUDT_Status.InvalidDataType := NOT (TypeOf(#iqv_Data) = TypeOfElements(#iqv_DataBuffer));

	END_REGION

	REGION 3 – Mode validation

	    // Set the mode invalid if selected mode isn't one of the following: W- Write, R - Read, C - Clear, S - Status
	    #tUDT_Status.InvalidMode := #ic_Mode <> 'W'
	    AND #ic_Mode <> 'R'
	    AND #ic_Mode <> 'C'
	    AND #ic_Mode <> 'S';

	END_REGION

	REGION 4 – The header settings checking

	    // The correct mode has been selected and data type is valid
	    IF (NOT #tUDT_Status.InvalidMode
	        AND NOT #tUDT_Status.InvalidDataType)
	    THEN

	        REGION 4.1 – The number of maximum FIFO entries validation

	            // Write the number of array's elements to FIFO header
	            #iqUDT_FifoHeader.MaxNrOfEntries := "FC_GetNrOfArrayEl"(#iqv_DataBuffer);

	            // Set the invalid maximum number of entries error
	            #tUDT_Status.InvalidMaxNrOfEntries := #iqUDT_FifoHeader.MaxNrOfEntries <= 0;

	        END_REGION

	        REGION 4.2 – The number of total FIFO entries validation

	            // Set the invalid total number of entries error
	            #tUDT_Status.InvalidTotalEntriesStored := #iqUDT_FifoHeader.TotalEntriesStored < 0        // The total number of entries is lower than 0
	            OR #iqUDT_FifoHeader.TotalEntriesStored > #iqUDT_FifoHeader.MaxNrOfEntries;               // The total number of entries is greater than the maximum number of entries

	        END_REGION

	        REGION 4.3 – The number of the next entry to write

	            // Set the invalid next entry to write
	            #tUDT_Status.InvalidNextEntryToWrite := #iqUDT_FifoHeader.NextEntryToWrite < 0            // The number of next entry to write is lower than 0
	            OR #iqUDT_FifoHeader.NextEntryToWrite >= #iqUDT_FifoHeader.MaxNrOfEntries;                // The number of next entry to write is greater or equal to the maximum number of entries

	        END_REGION

	        REGION 4.4 – The number of the next entry to read

	            // Set the invalid next entry to read
	            #tUDT_Status.InvalidNextEntryToRead := #iqUDT_FifoHeader.NextEntryToRead < 0              // The number of next entry to read is lower than 0
	            OR #iqUDT_FifoHeader.NextEntryToRead >= #iqUDT_FifoHeader.MaxNrOfEntries;                 // The number of next entry to read is greater or equal to the maximum nr of entries

	        END_REGION

	        REGION 4.5 – FIFO header validation summary

	            // Create collective header error
	            #tx_HeaderValid := NOT #tUDT_Status.InvalidMaxNrOfEntries
	            AND NOT #tUDT_Status.InvalidTotalEntriesStored
	            AND NOT #tUDT_Status.InvalidNextEntryToWrite
	            AND NOT #tUDT_Status.InvalidNextEntryToRead;

	        END_REGION

	    END_IF;

	END_REGION

	REGION 5 – Writing the data into the FIFO buffer

	    IF (#ic_Mode = 'W'                                                                          // Write mode selected
	        AND #tx_HeaderValid                                                                     // FIFO header valid
	        AND NOT #tUDT_Status.InvalidDataType)                                                  // Buffer data type valid
	    THEN


	        IF (#iqUDT_FifoHeader.TotalEntriesStored < #iqUDT_FifoHeader.MaxNrOfEntries)          // Checking total number of stored entries
	        THEN

	            // Move input data to FIFO data buffer
	            #ti_MoveBLKErrorCode := MOVE_BLK_VARIANT(SRC := #iqv_Data,
	                                                     COUNT := 1,
	                                                     SRC_INDEX := 0,
	                                                     DEST_INDEX := #iqUDT_FifoHeader.NextEntryToWrite,
	                                                     DEST => #iqv_DataBuffer);

	            // Increment the number of the next entry to write
	            #iqUDT_FifoHeader.NextEntryToWrite += 1;

	            // Increment the total number of stored entries
	            #iqUDT_FifoHeader.TotalEntriesStored += 1;


	            IF (#iqUDT_FifoHeader.NextEntryToWrite >= #iqUDT_FifoHeader.MaxNrOfEntries)       // Check the number of the next entry to write
	            THEN

	                #iqUDT_FifoHeader.NextEntryToWrite := 0;

	            END_IF;

	        ELSE

	            #tUDT_Status.FifoFull := TRUE;

	        END_IF;

	    END_IF;

	END_REGION

	REGION 6 – Reading the data from the FIFO data buffer

	    IF (#ic_Mode = 'R'                                                                  // Read mode selected
	        AND #tx_HeaderValid                                                             // FIFO header valid
	        AND NOT #tUDT_Status.InvalidDataType)                                           // Buffer data type valid
	    THEN

	        IF (#iqUDT_FifoHeader.TotalEntriesStored > 0)                                   // Checking total number of stored entries
	        THEN

	            // Move the FIFO data to the data output
	            #ti_MoveBLKErrorCode := MOVE_BLK_VARIANT(SRC := #iqv_DataBuffer,
	                                                     COUNT := 1,
	                                                     SRC_INDEX := #iqUDT_FifoHeader.NextEntryToRead,
	                                                     DEST_INDEX := 0,
	                                                     DEST => #iqv_Data);

	            // Increment the number of the next entry to read
	            #iqUDT_FifoHeader.NextEntryToRead += 1;

	            // Decrement the total number of stored entries
	            #iqUDT_FifoHeader.TotalEntriesStored -= 1;

	            IF (#iqUDT_FifoHeader.NextEntryToRead >= #iqUDT_FifoHeader.MaxNrOfEntries)  // Check the number of the next entry to read
	            THEN

	                #iqUDT_FifoHeader.NextEntryToRead := 0;

	            END_IF;

	        END_IF;

	    END_IF;

	END_REGION

	REGION 7 – Clearing the FIFO header

	    IF (#ic_Mode = 'C'                      // Clear mode selected
	        AND #tx_HeaderValid)                // FIFO header valid
	    THEN

	        #iqUDT_FifoHeader.TotalEntriesStored := 0;
	        #iqUDT_FifoHeader.NextEntryToWrite := 0;
	        #iqUDT_FifoHeader.NextEntryToRead := 0;

	    END_IF;

	END_REGION

	REGION 8 – FIFO management status update

	    IF (#tx_HeaderValid)                   // The header is valid
	    THEN

	        REGION 8.1 – FIFO Empty

	            // Set the FIFO empty status bit
	            #iqUDT_FifoHeader.Status.Empty := #iqUDT_FifoHeader.TotalEntriesStored = 0;

	        END_REGION

	        REGION 8.2 – FIFO Full

	            // Set the FIFO full status bit
	            #iqUDT_FifoHeader.Status.Full := #iqUDT_FifoHeader.TotalEntriesStored = #iqUDT_FifoHeader.MaxNrOfEntries;

	        END_REGION

	        REGION 8.3 – FIFO Pre-full

	            IF (#iqUDT_FifoHeader.TotalEntriesStored >= 0.9 * #iqUDT_FifoHeader.MaxNrOfEntries)       // Checking if the number of total stored entries is greater or equal to 90% of the max number of entries
	            THEN

	                // Set the FIFO pre-full status
	                #iqUDT_FifoHeader.Status.Prefull := TRUE;
	                #tUDT_Status.FifoPreFull := TRUE;

	            ELSE

	                #iqUDT_FifoHeader.Status.Prefull := FALSE;

	            END_IF;

	        END_REGION

	    END_IF;

	END_REGION

	REGION 9 – Status

	    REGION 9.1 – Common status update

	        // Collective error output
	        #qx_Error := NOT #tx_HeaderValid
	        OR #tUDT_Status.InvalidMode
	        OR #tUDT_Status.FifoFull
	        OR #tUDT_Status.InvalidDataType;

	        // Collective warning output
	        #qx_Warning := #tUDT_Status.FifoPreFull;

	    END_REGION

	    REGION 9.2 – Status update

	        // Update the outer status structure with internal status structure
	        #qUDT_Status := #tUDT_Status;

	    END_REGION

	END_REGION
END_FUNCTION

DATA_BLOCK "DB_GINDefault"
{ S7_Optimized_Access := 'TRUE' }
VERSION : 0.1
NON_RETAIN
   VAR
      GIN { ExternalAccessible := 'False'; ExternalVisible := 'False'; ExternalWritable := 'False'; S7_SetPoint := 'False'} : Array[1..20] of "UDT_GIN";   // GIN informations
   END_VAR


BEGIN

END_DATA_BLOCK

TYPE "UDT_ValveConfiguration"
VERSION : 0.1
   STRUCT
      ControlMode : Int := 1;   // 1 = Hold ix_open to keep qx_open active, 2 = detects rising edge on ix_Open to Open, ix_Close to Close
      ValveType : Int := 1;   // 1 = SEV, 2 = DEV
      CloseFeedBackExist { ExternalAccessible := 'False'; ExternalVisible := 'False'; ExternalWritable := 'False'} : Bool;   // Valve has a feed back that signals when fully cLosed
      OpenFeedBackExist { ExternalAccessible := 'False'; ExternalVisible := 'False'; ExternalWritable := 'False'} : Bool;   // Valve has a feed back that signals when fully Open
      OpenTime : Int;   // estimated open time, will trigger FTO if open feedback exist and not detected
      CloseTime : Int;   // estimated close time, will trigger FTC if close feedback exist and not detected
   END_STRUCT;

END_TYPE

FUNCTION "FC_WriteGIN" : Void
{ S7_Optimized_Access := 'TRUE' }
VERSION : 0.1
// ATTRIBUTES
// AUTO_NUMBER = True
// BLOCK_NUMBER = 31
// END_ATTRIBUTES
   VAR_INPUT
      ii_GIN : Int;   //    GIN number
      ii_PositionToWrite : Int;   //    Position in tracking array where to start writing GIN
      ii_NumberOfPositions : Int;   //    Number of positions to be written
      ix_Direction : Bool;   //    TRUE when positions in positive direction have to be written
   END_VAR

   VAR_IN_OUT
      iqa_TrackingData : Array[*] of Int;   //    Tracking data
   END_VAR

   VAR_TEMP
      ti_LCWritePosition : Int;   //    Loop counter
   END_VAR


BEGIN
	(*
	----------------------------------------------------------------------------------------

	Version history:
	Date        | Version   | Author        | Remark
	----------------------------------------------------------------------------------------
	27/02/2020  | 3.1       | L.Klar        | first release MHSE TIA 15.1
	21/02/2023  | 4.0       | F.Baten       | 4.0 Release TIA 17.5
	*)

	REGION 1 – GIN write

	    // Depending on the direction, a GIN is written into a specific number of tracking array positions.
	    #ti_LCWritePosition := 0;

	    IF #ix_Direction
	    THEN
	        FOR #ti_LCWritePosition := #ii_PositionToWrite TO #ii_PositionToWrite + #ii_NumberOfPositions - 1 BY 1 DO
	            #iqa_TrackingData[#ti_LCWritePosition] := #ii_GIN;
	        END_FOR;
	    ELSE
	        FOR #ti_LCWritePosition := #ii_PositionToWrite TO #ii_PositionToWrite - #ii_NumberOfPositions + 1 BY -1 DO
	            #iqa_TrackingData[#ti_LCWritePosition] := #ii_GIN;
	        END_FOR;
	    END_IF;

	END_REGION
END_FUNCTION

TYPE "UDT_PNNodeStatistics"
VERSION : 0.1
   STRUCT
      PNSlaveError : "UDT_EventStatistic";   // Statistics of a Profinet slave error
      PNSlaveNotOnline : "UDT_EventStatistic";   // Statistics of  Profinet slave not online
   END_STRUCT;

END_TYPE

FUNCTION_BLOCK "FB_ParcelLength"
{ S7_Optimized_Access := 'TRUE' }
VERSION : 0.1
// ATTRIBUTES
// AUTO_NUMBER = True
// BLOCK_NUMBER = 20
// END_ATTRIBUTES
   VAR_INPUT
      ii_PECPosition { ExternalAccessible := 'False'; ExternalVisible := 'False'; ExternalWritable := 'False'} : Int;   //    Photoeye position [cm]
      ii_Displacement { ExternalAccessible := 'False'; ExternalVisible := 'False'; ExternalWritable := 'False'} : Int;   //    Displacement [cm]
      ix_LengthMeasurementEnable { ExternalAccessible := 'False'; ExternalVisible := 'False'; ExternalWritable := 'False'} : Bool;   //    Length measurement enable
      ix_GapMeasurementEnable { ExternalAccessible := 'False'; ExternalVisible := 'False'; ExternalWritable := 'False'} : Bool;   //    Gap measurement enable
   END_VAR

   VAR_IN_OUT
      iqa_TrackingData : Array[*] of Int;   //    Tracking data
   END_VAR

   VAR
      sR_TRIG_Data {InstructionName := 'R_TRIG'; LibVersion := '1.0'; ExternalAccessible := 'False'; ExternalVisible := 'False'; ExternalWritable := 'False'; S7_SetPoint := 'False'} : R_TRIG;   //    Data rising edge for length and gap measurements
      sF_TRIG_Data {InstructionName := 'F_TRIG'; LibVersion := '1.0'; ExternalAccessible := 'False'; ExternalVisible := 'False'; ExternalWritable := 'False'; S7_SetPoint := 'False'} : F_TRIG;   //    Data falling edge for length and gap measurements
      si_Length { ExternalAccessible := 'False'; ExternalVisible := 'False'; ExternalWritable := 'False'} : Int;   //    Parcel length
      si_Gap { ExternalAccessible := 'False'; ExternalVisible := 'False'; ExternalWritable := 'False'} : Int;   //    Gap distance
      si_GIN { ExternalAccessible := 'False'; ExternalVisible := 'False'; ExternalWritable := 'False'} : Int;   //    GIN number of current measured parcel
      si_OldGIN { ExternalAccessible := 'False'; ExternalVisible := 'False'; ExternalWritable := 'False'} : Int;   //    GIN number of previous mesured parcel
   END_VAR

   VAR CONSTANT
      ci_Overflow : Int := 32767;   //    Integer overflow value
   END_VAR


BEGIN
	(*
	----------------------------------------------------------------------------------------

	Version history:
	Date        | Version   | Author        | Remark
	----------------------------------------------------------------------------------------
	21/02/2020  | 3.1       | L.Klar        | first release MHSE TIA 15.1
	21/02/2023  | 4.0       | F.Baten       | 4.0 Release TIA 17.5
	*)

	REGION 1 – Data triggers

	    // Triggers to detect front and end of data

	    #sR_TRIG_Data(CLK := #iqa_TrackingData[#ii_PECPosition] > 0);
	    #sF_TRIG_Data(CLK := #iqa_TrackingData[#ii_PECPosition] > 0);

	END_REGION

	REGION 2 – Length counter

	    //  Length is counted from a displacement, when data is available
	    //
	    IF (#iqa_TrackingData[#ii_PECPosition] > 0
	        AND #ix_LengthMeasurementEnable
	        AND #si_Length < #ci_Overflow)

	    THEN
	        #si_Length += #ii_Displacement;
	    END_IF;

	END_REGION

	REGION 3 – Gap counter

	    //  Gap is counted from a displacement, when data isn't available
	    IF (#iqa_TrackingData[#ii_PECPosition] = 0
	        AND #ix_GapMeasurementEnable
	        AND #si_Gap < #ci_Overflow)
	    THEN
	        #si_Gap += #ii_Displacement;
	    END_IF;

	END_REGION

	REGION 4 – Parcel GIN

	    IF (#sR_TRIG_Data.Q AND
	        (#ix_LengthMeasurementEnable OR #ix_GapMeasurementEnable))
	    THEN
	        #si_GIN := #iqa_TrackingData[#ii_PECPosition];
	    END_IF;

	END_REGION

	REGION 5 – Write length into a GIN record

	    IF (#sF_TRIG_Data.Q)
	    THEN

	        IF #ix_LengthMeasurementEnable OR #ix_GapMeasurementEnable THEN
	            #si_OldGIN := #si_GIN;
	        END_IF;

	        IF (#si_GIN > 0
	            AND ABS(#si_Length) > 0
	            AND #ix_LengthMeasurementEnable)
	        THEN
	            "DB_GIN".GIN[#si_GIN].General.Length := ABS(#si_Length) - 1;
	            #si_Length := 0;
	        ELSE
	            #si_Length := 0;
	        END_IF;
	    END_IF;

	END_REGION

	REGION 6 – Write GIN into a GIN record

	    IF (#sR_TRIG_Data.Q)
	    THEN
	        IF (#si_OldGIN > 0
	            AND #si_GIN > 0
	            AND #si_Gap <> 0
	            AND #si_OldGIN <> #si_GIN
	            AND #ix_GapMeasurementEnable)
	        THEN
	            IF (#ii_Displacement > 0)
	            THEN
	                "DB_GIN".GIN[#si_GIN].General.LeadingGap := ABS(#si_Gap) - 1;
	                "DB_GIN".GIN[#si_OldGIN].General.TrailingGap := "DB_GIN".GIN[#si_GIN].General.LeadingGap;
	                #si_Gap := 0;
	            ELSIF (#ii_Displacement < 0)
	            THEN
	                "DB_GIN".GIN[#si_OldGIN].General.LeadingGap := ABS(#si_Gap - 1);
	                "DB_GIN".GIN[#si_GIN].General.TrailingGap := "DB_GIN".GIN[#si_OldGIN].General.LeadingGap;
	                #si_Gap := 0;
	            END_IF;
	        ELSE
	            #si_Gap := 0;
	        END_IF;
	    END_IF;

	END_REGION
END_FUNCTION_BLOCK

TYPE "UDT_ValveStatus"
TITLE = UDT_ConveyorStatus
VERSION : 0.1
//User-defined structure of FB_Conveyor function block status.
   STRUCT
      Status { ExternalWritable := 'False'} : Int;   // Status number
      Specific { ExternalWritable := 'False'} : Struct
         Opening { ExternalAccessible := 'False'; ExternalVisible := 'False'; ExternalWritable := 'False'} : Bool;   // Valve is opening
         Opened { ExternalAccessible := 'False'; ExternalVisible := 'False'; ExternalWritable := 'False'} : Bool;   // Valve in Open position
         Closing { ExternalAccessible := 'False'; ExternalVisible := 'False'; ExternalWritable := 'False'} : Bool;   // Valve is closing
         Closed { ExternalAccessible := 'False'; ExternalVisible := 'False'; ExternalWritable := 'False'} : Bool;   // Valve in Closed position
         FailToOpen { ExternalAccessible := 'False'; ExternalVisible := 'False'; ExternalWritable := 'False'} : Bool;   // Fail to open / extend
         FailToClose { ExternalAccessible := 'False'; ExternalVisible := 'False'; ExternalWritable := 'False'} : Bool;   // Fail to close / retract
         AirPressureLost { ExternalAccessible := 'False'; ExternalVisible := 'False'; ExternalWritable := 'False'} : Bool;   // No air pressure
         ConfigurationError { ExternalAccessible := 'False'; ExternalVisible := 'False'; ExternalWritable := 'False'} : Bool;   // Configuration is not set correctly
      END_STRUCT;
   END_STRUCT;

END_TYPE

TYPE "UDT_AixPlcFullControllerConfiguration"
TITLE = UDT_VFD_Configuration
VERSION : 0.1
//User-defined structure oparameters.
   STRUCT
      AixContrlPNDeviceName { ExternalAccessible := 'False'; ExternalVisible := 'False'; ExternalWritable := 'False'} : String;   // Ai2's Controller Profinet device name
      Motor { ExternalAccessible := 'False'; ExternalVisible := 'False'; ExternalWritable := 'False'} : Struct
         RampUpTime { ExternalAccessible := 'False'; ExternalVisible := 'False'; ExternalWritable := 'False'} : UDInt := 100;   // Ramp up time for monitoring starting [ms]
         RampDownTime { ExternalAccessible := 'False'; ExternalVisible := 'False'; ExternalWritable := 'False'} : UDInt := 100;   // Ramp up time for monitoring stopping [ms]
         SpeedSetpointWindow { ExternalAccessible := 'False'; ExternalVisible := 'False'; ExternalWritable := 'False'} : Int := 5;   // Speed setpoint window (tolerance) [mm/s]
         Ratio { ExternalAccessible := 'False'; ExternalVisible := 'False'; ExternalWritable := 'False'} : Real := 1.0;   // Ratio conveyor roller to driven roller
         DirectionReversal { ExternalAccessible := 'False'; ExternalVisible := 'False'; ExternalWritable := 'False'} : Bool;   // True = direction will be reversed
         InterlockFwd { ExternalAccessible := 'False'; ExternalVisible := 'False'; ExternalWritable := 'False'} : Bool := TRUE;   // False = running in forward direction is not possible / allowed
         InterlockRvs { ExternalAccessible := 'False'; ExternalVisible := 'False'; ExternalWritable := 'False'} : Bool;   // False = running in reverse direction is not possible / allowed
         MotorExist { ExternalAccessible := 'False'; ExternalVisible := 'False'; ExternalWritable := 'False'} : Bool;   // True = Motor output connected
      END_STRUCT;
   END_STRUCT;

END_TYPE

